// Auto Bagger 
GVL_IO.BG_YFillerTrigger					:= BYTE_TO_BOOL(GVL_IO.OutputsFromHMI[91]);
IF (STATUS.BaggerPrintCmd = 1) THEN 
	MAIN.fbEL6001.M_PrintLabel(isPremium := FALSE);  
    STATUS.BaggerPrintCmd := 0;
    (* We now have a separate button for Clear Out Chute Counts
    Config.PremiumCount1 := 0;
    Config.PremiumCount2 := 0;
	Config.GoodCount1 := 0;
	Config.GoodCount2 := 0;
    *) 
 END_IF // print label trigger from HMI

GVL_IO.BG_YCloseChute1 := BYTE_TO_BOOL(GVL_IO.OutputsFromHMI[92]); 	
GVL_IO.BG_YOpenChute1  := BYTE_TO_BOOL(GVL_IO.OutputsFromHMI[93]);  	
GVL_IO.BG_YCloseChute2 := BYTE_TO_BOOL(GVL_IO.OutputsFromHMI[94]); 	
GVL_IO.BG_YOpenChute2  := BYTE_TO_BOOL(GVL_IO.OutputsFromHMI[95]); 	
GVL_IO.BG_YCloseChute3 := BYTE_TO_BOOL(GVL_IO.OutputsFromHMI[96]); 	
GVL_IO.BG_YOpenChute3  := BYTE_TO_BOOL(GVL_IO.OutputsFromHMI[97]); 	
GVL_IO.BG_YCloseChute4 := BYTE_TO_BOOL(GVL_IO.OutputsFromHMI[98]); 	
GVL_IO.BG_YOpenChute4  := BYTE_TO_BOOL(GVL_IO.OutputsFromHMI[99]); 	






// Reject Unload
GVL_IO.RJ_YRejectPushExtend				:= BYTE_TO_BOOL(GVL_IO.OutputsFromHMI[101]); 	
GVL_IO.RJ_YRejectPushRetract			:= BYTE_TO_BOOL(GVL_IO.OutputsFromHMI[102]); 	
//GVL_IO.RJ_YPalletReleaseExtend			:= BYTE_TO_BOOL(GVL_IO.OutputsFromHMI[103]); 	
//GVL_IO.RJ_YPalletReleaseRetract			:= BYTE_TO_BOOL(GVL_IO.OutputsFromHMI[104]); 	
GVL_IO.RJ_YPalletHoldDownExtend_Home			:= BYTE_TO_BOOL(GVL_IO.OutputsFromHMI[105]); 	
GVL_IO.RJ_YPalletHoldDownRetract_Engage		:= BYTE_TO_BOOL(GVL_IO.OutputsFromHMI[106]); 	
                                                                                        
// Main Control System

GVL_IO.MC_YStackLightYellow				:= BYTE_TO_BOOL(GVL_IO.OutputsFromHMI[111]);
GVL_IO.MC_YStackLightRed				:= BYTE_TO_BOOL(GVL_IO.OutputsFromHMI[112]);
GVL_IO.MC_YStackLightGreen				:= BYTE_TO_BOOL(GVL_IO.OutputsFromHMI[113]);
                                        

// Prime Mover 
GVL_IO.MM_YEnableMagneMotion           := BYTE_TO_BOOL(GVL_IO.OutputsFromHMI[121]);

END_FUNCTION_BLOCK

// ---- POUs/FrameworkPOUs/PrepareInputsDataStructureForHMI.TcPOU
// Fill up the appropriate data structure to send input data to the HMI 
FUNCTION_BLOCK FINAL PrepareInputsDataStructureForHMI
VAR_INPUT
END_VAR
VAR_OUTPUT
END_VAR
VAR
	UL_X: INT;
END_VAR

memset(ADR(GVL_IO.InputsForHMI[1]),0,SIZEOF(GVL_IO.InputsForHMI)); //clear out the input array

// Load Station
GVL_IO.InputsForHMI[1] := 	BOOL_TO_BYTE(GVL_IO.LD_XPalletHoldRetractEngage);
GVL_IO.InputsForHMI[2] := 	BOOL_TO_BYTE(GVL_IO.LD_XPalletHoldDownExtendHome);
GVL_IO.InputsForHMI[3] := 	BOOL_TO_BYTE(GVL_IO.LD_XPalletReleaseHome);
GVL_IO.InputsForHMI[4] := 	BOOL_TO_BYTE(GVL_IO.LD_XPalletReleaseExtended);
GVL_IO.InputsForHMI[15] := 	BOOL_TO_BYTE(GVL_IO.LD_XPalletCloseExtended_1_2);
GVL_IO.InputsForHMI[16] := 	BOOL_TO_BYTE(GVL_IO.LD_XPalletCloseExtended_3_4);
GVL_IO.InputsForHMI[17] := 	BOOL_TO_BYTE(GVL_IO.LD_XPalletCloseRetracted_1_2);
GVL_IO.InputsForHMI[18] := 	BOOL_TO_BYTE(GVL_IO.LD_XPalletCloseRetracted_3_4);

// Yushin Robot 
GVL_IO.InputsForHMI[5] := 	BOOL_TO_BYTE(GVL_IO.YU_XPrepareToLoad);
GVL_IO.InputsForHMI[6] := 	BOOL_TO_BYTE(GVL_IO.YU_XToolUp);           
GVL_IO.InputsForHMI[7] := 	BOOL_TO_BYTE(GVL_IO.YU_XToolDown);
GVL_IO.InputsForHMI[8] := 	BOOL_TO_BYTE(GVL_IO.YU_XLocBit0);
GVL_IO.InputsForHMI[9] := 	BOOL_TO_BYTE(GVL_IO.YU_XLocBit1);

// Burnoff
GVL_IO.InputsForHMI[11] := 	BOOL_TO_BYTE(GVL_IO.BU_XAlarm);

// Ionizer 
GVL_IO.InputsForHMI[12] := 	BOOL_TO_BYTE(GVL_IO.IZ_XIonAlarm);
GVL_IO.InputsForHMI[13] := 	BOOL_TO_BYTE(GVL_IO.IZ_XConditionAlarm);
GVL_IO.InputsForHMI[14] := 	BOOL_TO_BYTE(GVL_IO.IZ_XAlarm);
// borrowing 15,16,17,18 for Load Station Pallet Close inputs
// Vision
GVL_IO.InputsForHMI[21] := 	BOOL_TO_BYTE(GVL_IO.VS_XToolingLocationUpper);
GVL_IO.InputsForHMI[22] := 	BOOL_TO_BYTE(GVL_IO.VS_XRun);
GVL_IO.InputsForHMI[23] := 	BOOL_TO_BYTE(GVL_IO.VS_XReady1);
GVL_IO.InputsForHMI[24] := 	BOOL_TO_BYTE(GVL_IO.VS_XReady2);
GVL_IO.InputsForHMI[25] := 	BOOL_TO_BYTE(GVL_IO.VS_XReady3);
GVL_IO.InputsForHMI[26] := 	BOOL_TO_BYTE(GVL_IO.VS_XReady4);
GVL_IO.InputsForHMI[27] := 	BOOL_TO_BYTE(GVL_IO.VS_XCam1JudgeVal);
GVL_IO.InputsForHMI[28] := 	BOOL_TO_BYTE(GVL_IO.VS_XCam2JudgeVal);
GVL_IO.InputsForHMI[29] := 	BOOL_TO_BYTE(GVL_IO.VS_XCam3JudgeVal);
GVL_IO.InputsForHMI[30] := 	BOOL_TO_BYTE(GVL_IO.VS_XCam4JudgeVal);
GVL_IO.InputsForHMI[92] := 	BOOL_TO_BYTE(GVL_IO.VS_XPartEmpty);
GVL_IO.InputsForHMI[93] :=  BOOL_TO_BYTE(GVL_IO.VS_XToolingLocationLower);
GVL_IO.InputsForHMI[94] :=  BOOL_TO_BYTE(GVL_IO.VS_XPartPresentBeforeVision);

// Piston Insert 
GVL_IO.InputsForHMI[31] := 	BOOL_TO_BYTE(GVL_IO.PI_XPalletHoldDownHome);
GVL_IO.InputsForHMI[32] := 	BOOL_TO_BYTE(GVL_IO.PI_XPalletHoldDownExtended);
GVL_IO.InputsForHMI[33] := 	BOOL_TO_BYTE(GVL_IO.PI_XPistonPresentEscapement);
GVL_IO.InputsForHMI[34] := 	BOOL_TO_BYTE(GVL_IO.PI_XEscapementAtInsertLoc);
GVL_IO.InputsForHMI[35] := 	BOOL_TO_BYTE(GVL_IO.PI_XEscapementAtBowl);
GVL_IO.InputsForHMI[36] := 	BOOL_TO_BYTE(GVL_IO.PI_XToolAt55_10_Barrel);
GVL_IO.InputsForHMI[37] := 	BOOL_TO_BYTE(GVL_IO.PI_XToolAt3_30_Barrel);
GVL_IO.InputsForHMI[38] := 	BOOL_TO_BYTE(GVL_IO.PI_XBarrelHoldDownHome);
GVL_IO.InputsForHMI[39] := 	BOOL_TO_BYTE(GVL_IO.PI_XBarrelHoldDownExtended);

//GVL_IO.InputsForHMI[40] := 1;
GVL_IO.InputsForHMI[40] := BOOL_TO_BYTE(GVL_IO.PI_XMtrOUT0);
GVL_IO.InputsForHMI[41] := BOOL_TO_BYTE(GVL_IO.PI_XMtrOUT1);
GVL_IO.InputsForHMI[42] := BOOL_TO_BYTE(GVL_IO.PI_XMtrBusy);
GVL_IO.InputsForHMI[43] := BOOL_TO_BYTE(GVL_IO.PI_XMtrServoEnabled);
GVL_IO.InputsForHMI[44] := BOOL_TO_BYTE(GVL_IO.PI_XMtrServoHomed);
GVL_IO.InputsForHMI[45] := BOOL_TO_BYTE(GVL_IO.PI_XMtrMoveCompl);
GVL_IO.InputsForHMI[46] := BOOL_TO_BYTE(GVL_IO.PI_XMtrEStopped);
GVL_IO.InputsForHMI[47] := BOOL_TO_BYTE(GVL_IO.PI_XMtrAlarm);


// Cap Insert

GVL_IO.InputsForHMI[56] := 	BOOL_TO_BYTE(GVL_IO.CP_XPalletHoldDownHome);
GVL_IO.InputsForHMI[57] := 	BOOL_TO_BYTE(GVL_IO.CP_XPalletHoldDownExtended);
GVL_IO.InputsForHMI[58] := 	BOOL_TO_BYTE(GVL_IO.CP_XCapSlideRetracted);
GVL_IO.InputsForHMI[59] := 	BOOL_TO_BYTE(GVL_IO.CP_XCapSlideExtended);


// Unload 

GVL_IO.InputsForHMI[77] :=  BOOL_TO_BYTE(GVL_IO.UL_1_XPalletHoldDownRetracted_Engaged);
GVL_IO.InputsForHMI[78] :=  BOOL_TO_BYTE(GVL_IO.UL_1_XPalletHoldDownExtended_Home);
GVL_IO.InputsForHMI[79] := 	BOOL_TO_BYTE(GVL_IO.UL_1_XBarrelPresent);
GVL_IO.InputsForHMI[80] :=  BOOL_TO_BYTE(GVL_IO.UL_2_XPalletHoldDownRetracted_Engaged);
GVL_IO.InputsForHMI[81] :=  BOOL_TO_BYTE(GVL_IO.UL_2_XPalletHoldDownExtended_Home);
GVL_IO.InputsForHMI[82] := 	BOOL_TO_BYTE(GVL_IO.UL_2_XBarrelPresent);
GVL_IO.InputsForHMI[83] :=  BOOL_TO_BYTE(GVL_IO.UL_3_XPalletHoldDownRetracted_Engaged);
GVL_IO.InputsForHMI[84] :=  BOOL_TO_BYTE(GVL_IO.UL_3_XPalletHoldDownExtended_Home);
GVL_IO.InputsForHMI[85] := 	BOOL_TO_BYTE(GVL_IO.UL_3_XBarrelPresent);
GVL_IO.InputsForHMI[86] :=  BOOL_TO_BYTE(GVL_IO.UL_4_XPalletHoldDownRetracted_Engaged);
GVL_IO.InputsForHMI[87] :=  BOOL_TO_BYTE(GVL_IO.UL_4_XPalletHoldDownExtended_Home);
GVL_IO.InputsForHMI[88] := 	BOOL_TO_BYTE(GVL_IO.UL_4_XBarrelPresent);


// bagger
GVL_IO.InputsForHMI[91] := 	BOOL_TO_BYTE(GVL_IO.BG_XBaggerBusy);
//borrowing 92 for vision
// borrowing 93 for vision
// borrow 94 for vision
GVL_IO.InputsForHMI[115] := 	BOOL_TO_BYTE(GVL_IO.BG_XBagsLow);
GVL_IO.InputsForHMI[116] := 	BOOL_TO_BYTE(GVL_IO.BG_XBaggerOKNoFault);
GVL_IO.InputsForHMI[117] := 	BOOL_TO_BYTE(GVL_IO.BG_XBaggerWaitingForLabel);
GVL_IO.InputsForHMI[118] := 	BOOL_TO_BYTE(GVL_IO.BG_XBaggerReadyForFiller);


GVL_IO.InputsForHMI[95] := 	BOOL_TO_BYTE(GVL_IO.BG_XChute1Closed);
GVL_IO.InputsForHMI[96] := 	BOOL_TO_BYTE(GVL_IO.BG_XChute1Open);
GVL_IO.InputsForHMI[97] := 	BOOL_TO_BYTE(GVL_IO.BG_XChute2Closed);
GVL_IO.InputsForHMI[98] := 	BOOL_TO_BYTE(GVL_IO.BG_XChute2Open);
GVL_IO.InputsForHMI[99] := 	BOOL_TO_BYTE(GVL_IO.BG_XChute3Closed);
GVL_IO.InputsForHMI[100] := BOOL_TO_BYTE(GVL_IO.BG_XChute3Open);  
GVL_IO.InputsForHMI[108] := BOOL_TO_BYTE(GVL_IO.BG_XChute4Closed);
GVL_IO.InputsForHMI[109] := BOOL_TO_BYTE(GVL_IO.BG_XChute4Open);  



// Reject Station 
GVL_IO.InputsForHMI[101] := 	BOOL_TO_BYTE(GVL_IO.RJ_XRejectCylinderHome);
GVL_IO.InputsForHMI[102] := 	BOOL_TO_BYTE(GVL_IO.RJ_XRejectCylinderExtended);
//GVL_IO.InputsForHMI[103] := 	BOOL_TO_BYTE(GVL_IO.RJ_XPalletReleaseHome);
//GVL_IO.InputsForHMI[104] := 	BOOL_TO_BYTE(GVL_IO.RJ_XPalletReleaseExtended);
GVL_IO.InputsForHMI[105] := 	BOOL_TO_BYTE(GVL_IO.RJ_XPartPresent);
GVL_IO.InputsForHMI[106] := 	BOOL_TO_BYTE(GVL_IO.RJ_XPalletHoldDownRetracted_Engaged);
GVL_IO.InputsForHMI[107] := 	BOOL_TO_BYTE(GVL_IO.RJ_XPalletHoldDownExtended_Home);
// borrowing 108 and 109 for Autobagger inputs

// Main Control System
GVL_IO.InputsForHMI[111] := 	BOOL_TO_BYTE(GVL_IO.MC_XAirPressureOK);
GVL_IO.InputsForHMI[112] := 	BOOL_TO_BYTE(GVL_IO.MC_XStartPB);
GVL_IO.InputsForHMI[113] := 	BOOL_TO_BYTE(GVL_IO.MC_XStopPB);
GVL_IO.InputsForHMI[114] := 	BOOL_TO_BYTE(GVL_IO.MC_NotEStopped);
// borrowing 115,116,117,118 for bagger inputs

END_FUNCTION_BLOCK

// ---- POUs/FrameworkPOUs/PrepareOutputsDataStructureForHMI.TcPOU
// Fill up the appropriate data structure to send input data to the HMI 
FUNCTION_BLOCK FINAL PrepareOutputsDataStructureForHMI
VAR_INPUT
END_VAR
VAR_OUTPUT
END_VAR
VAR
END_VAR

memset(ADR(GVL_IO.OutputsForHMI[1]),0,SIZEOF(GVL_IO.InputsForHMI)); //clear out the output array

// Load Position Outputs 

GVL_IO.OutputsForHMI[1] 	:= BOOL_TO_BYTE(GVL_IO.LD_YPalletHoldDownRetractEngage);
GVL_IO.OutputsForHMI[2] 	:= BOOL_TO_BYTE(GVL_IO.LD_YPalletHoldDownExtendHome);
GVL_IO.OutputsForHMI[3] 	:= BOOL_TO_BYTE(GVL_IO.LD_YPalletReleaseExtend);
GVL_IO.OutputsForHMI[4] 	:= BOOL_TO_BYTE(GVL_IO.LD_YPalletReleaseRetract);
GVL_IO.OutputsForHMI[8]     := BOOL_TO_BYTE(GVL_IO.LD_YPalletCloseExtend);
GVL_IO.OutputsForHMI[9]     := BOOL_TO_BYTE(GVL_IO.LD_YPalletCloseRetract);

// Yushin Robot Interface Outputs

GVL_IO.OutputsForHMI[5] 	:= BOOL_TO_BYTE(GVL_IO.YU_YOkToLoad);
GVL_IO.OutputsForHMI[6] 	:= BOOL_TO_BYTE(GVL_IO.YU_YAckPartsHeld);
GVL_IO.OutputsForHMI[10]    := BOOL_TO_BYTE(GVL_IO.YU_YIMBADIsOK);

//Ionizer Outputs

GVL_IO.OutputsForHMI[7] 	:= BOOL_TO_BYTE(GVL_IO.IZ_YInterrupt);
//GVL_IO.OutputsForHMI[8]     := BOOL_TO_BYTE(GVL_IO.IZ_YIonizerAirON);
//GVL_IO.OutputsForHMI[9]     := BOOL_TO_BYTE(GVL_IO.IZ_YIonizerAirOFF);
// give 10 to Yushin

// Vision
GVL_IO.OutputsForHMI[21] 	:= BOOL_TO_BYTE(GVL_IO.VS_YBarrelLED);
GVL_IO.OutputsForHMI[22] 	:= BOOL_TO_BYTE(GVL_IO.VS_YCmdRequest);
GVL_IO.OutputsForHMI[23] 	:= BOOL_TO_BYTE(GVL_IO.VS_YResultAck);
GVL_IO.OutputsForHMI[24] 	:= BOOL_TO_BYTE(GVL_IO.VS_YErrorReset);
GVL_IO.OutputsForHMI[25] 	:= BOOL_TO_BYTE(GVL_IO.VS_YTrigger1);
GVL_IO.OutputsForHMI[26] 	:= BOOL_TO_BYTE(GVL_IO.VS_YTrigger2);
GVL_IO.OutputsForHMI[27] 	:= BOOL_TO_BYTE(GVL_IO.VS_YTrigger3);
GVL_IO.OutputsForHMI[28] 	:= BOOL_TO_BYTE(GVL_IO.VS_YTrigger4);


// Piston Insert 
GVL_IO.OutputsForHMI[31] 	:= BOOL_TO_BYTE(GVL_IO.PI_YPalletHoldDownExtend);
GVL_IO.OutputsForHMI[32] 	:= BOOL_TO_BYTE(GVL_IO.PI_YPalletHoldDownRetract);
GVL_IO.OutputsForHMI[33] 	:= BOOL_TO_BYTE(GVL_IO.PI_YEscapementToBowl);
GVL_IO.OutputsForHMI[34] 	:= BOOL_TO_BYTE(GVL_IO.PI_YEscapementToWork);
GVL_IO.OutputsForHMI[35] 	:= BOOL_TO_BYTE(GVL_IO.PI_YBarrelBackupExtend);
GVL_IO.OutputsForHMI[36] 	:= BOOL_TO_BYTE(GVL_IO.PI_YBarrelBackupRetract);
GVL_IO.OutputsForHMI[37] 	:= BOOL_TO_BYTE(GVL_IO.PI_YPistonBowlON);
GVL_IO.OutputsForHMI[38] 	:= BOOL_TO_BYTE(GVL_IO.PI_YPistonBowlOFF);

GVL_IO.OutputsForHMI[40] 	:= BOOL_TO_BYTE(GVL_IO.PI_YMtrStepSelectIN0);
GVL_IO.OutputsForHMI[41] 	:= BOOL_TO_BYTE(GVL_IO.PI_YMtrStepSelectIN1);
GVL_IO.OutputsForHMI[42] 	:= BOOL_TO_BYTE(GVL_IO.PI_YMtrStepSelectIN2);
GVL_IO.OutputsForHMI[43] 	:= BOOL_TO_BYTE(GVL_IO.PI_YMtrHoldMove);
GVL_IO.OutputsForHMI[44] 	:= BOOL_TO_BYTE(GVL_IO.PI_YMtrSetEnable);
GVL_IO.OutputsForHMI[45] 	:= BOOL_TO_BYTE(GVL_IO.PI_YMtrDriveStepTrigger);
GVL_IO.OutputsForHMI[46] 	:= BOOL_TO_BYTE(GVL_IO.PI_YMtrReset);
GVL_IO.OutputsForHMI[47] 	:= BOOL_TO_BYTE(GVL_IO.PI_YMtrGoHome);
GVL_IO.OutputsForHMI[48] 	:= BOOL_TO_BYTE(GVL_IO.PI_YMtrJogNeg);
GVL_IO.OutputsForHMI[49] 	:= BOOL_TO_BYTE(GVL_IO.PI_YMtrJogPos);
GVL_IO.OutputsForHMI[50] 	:= BOOL_TO_BYTE(GVL_IO.PI_YMtrSwitchJogInch);
// Cap Insert 

GVL_IO.OutputsForHMI[57] 	:= BOOL_TO_BYTE(GVL_IO.CP_YCapSlideExtend);
GVL_IO.OutputsForHMI[58] 	:= BOOL_TO_BYTE(GVL_IO.CP_YCapSlideRetract);
GVL_IO.OutputsForHMI[59] 	:= BOOL_TO_BYTE(GVL_IO.CP_YPalletHoldDownExtend);
GVL_IO.OutputsForHMI[60] 	:= BOOL_TO_BYTE(GVL_IO.CP_YPalletHoldDownRetract);


// Good Unload Outputs
 
GVL_IO.OutputsForHMI[71] 	:= BOOL_TO_BYTE(GVL_IO.UL_1_YPalletHoldDownExtend_Home);
GVL_IO.OutputsForHMI[72] 	:= BOOL_TO_BYTE(GVL_IO.UL_1_YPalletHoldDownRetract_Engage);
GVL_IO.OutputsForHMI[73] 	:= BOOL_TO_BYTE(GVL_IO.UL_2_YPalletHoldDownExtend_Home);
GVL_IO.OutputsForHMI[74] 	:= BOOL_TO_BYTE(GVL_IO.UL_2_YPalletHoldDownRetract_Engage);
GVL_IO.OutputsForHMI[75] 	:= BOOL_TO_BYTE(GVL_IO.UL_3_YPalletHoldDownExtend_Home);
GVL_IO.OutputsForHMI[76] 	:= BOOL_TO_BYTE(GVL_IO.UL_3_YPalletHoldDownRetract_Engage);
GVL_IO.OutputsForHMI[77] 	:= BOOL_TO_BYTE(GVL_IO.UL_4_YPalletHoldDownExtend_Home);   
GVL_IO.OutputsForHMI[78] 	:= BOOL_TO_BYTE(GVL_IO.UL_4_YPalletHoldDownRetract_Engage);

GVL_IO.OutputsForHMI[79] 	:= BOOL_TO_BYTE(GVL_IO.UL_1_YRejectPushExtend);
GVL_IO.OutputsForHMI[80] 	:= BOOL_TO_BYTE(GVL_IO.UL_2_YRejectPushExtend);
GVL_IO.OutputsForHMI[81] 	:= BOOL_TO_BYTE(GVL_IO.UL_3_YRejectPushExtend);
GVL_IO.OutputsForHMI[82] 	:= BOOL_TO_BYTE(GVL_IO.UL_4_YRejectPushExtend);

GVL_IO.OutputsForHMI[83] 	:= BOOL_TO_BYTE(GVL_IO.UL_1_YRejectPushRetract);
GVL_IO.OutputsForHMI[84] 	:= BOOL_TO_BYTE(GVL_IO.UL_2_YRejectPushRetract);
GVL_IO.OutputsForHMI[85] 	:= BOOL_TO_BYTE(GVL_IO.UL_3_YRejectPushRetract);
GVL_IO.OutputsForHMI[86] 	:= BOOL_TO_BYTE(GVL_IO.UL_4_YRejectPushRetract);




// Auto Bagger 
GVL_IO.OutputsForHMI[91] 	:= 	BOOL_TO_BYTE(GVL_IO.BG_YFillerTrigger);
GVL_IO.OutputsForHMI[92] 	:= 	BOOL_TO_BYTE(GVL_IO.BG_YCloseChute1);
GVL_IO.OutputsForHMI[93] 	:= 	BOOL_TO_BYTE(GVL_IO.BG_YOpenChute1);
GVL_IO.OutputsForHMI[94] 	:= 	BOOL_TO_BYTE(GVL_IO.BG_YCloseChute2);
GVL_IO.OutputsForHMI[95] 	:= 	BOOL_TO_BYTE(GVL_IO.BG_YOpenChute2);
GVL_IO.OutputsForHMI[96] 	:= 	BOOL_TO_BYTE(GVL_IO.BG_YCloseChute3);
GVL_IO.OutputsForHMI[97] 	:= 	BOOL_TO_BYTE(GVL_IO.BG_YOpenChute3);
GVL_IO.OutputsForHMI[98] 	:= 	BOOL_TO_BYTE(GVL_IO.BG_YCloseChute4);
GVL_IO.OutputsForHMI[99] 	:= 	BOOL_TO_BYTE(GVL_IO.BG_YOpenChute4);



// Reject Unload
GVL_IO.OutputsForHMI[101] 	:= BOOL_TO_BYTE(GVL_IO.RJ_YRejectPushExtend);
GVL_IO.OutputsForHMI[102] 	:= BOOL_TO_BYTE(GVL_IO.RJ_YRejectPushRetract);
//GVL_IO.OutputsForHMI[103] 	:= BOOL_TO_BYTE(GVL_IO.RJ_YPalletReleaseExtend);
//GVL_IO.OutputsForHMI[104] 	:= BOOL_TO_BYTE(GVL_IO.RJ_YPalletReleaseRetract);
GVL_IO.OutputsForHMI[105] 	:= BOOL_TO_BYTE(GVL_IO.RJ_YPalletHoldDownExtend_Home);
GVL_IO.OutputsForHMI[106] 	:= BOOL_TO_BYTE(GVL_IO.RJ_YPalletHoldDownRetract_Engage);

// Main Control System

GVL_IO.OutputsForHMI[111] 	:= BOOL_TO_BYTE(GVL_IO.MC_YStackLightYellow);
GVL_IO.OutputsForHMI[112] 	:= BOOL_TO_BYTE(GVL_IO.MC_YStackLightRed);
GVL_IO.OutputsForHMI[113] 	:= BOOL_TO_BYTE(GVL_IO.MC_YStackLightGreen);



// Prime Mover 
GVL_IO.OutputsForHMI[121] 	:= BOOL_TO_BYTE(GVL_IO.MM_YEnableMagneMotion);

END_FUNCTION_BLOCK

// ---- POUs/FrameworkPOUs/SetOutputsToFieldBus.TcPOU
// Setup the appropriate output from the outputs  coming from the logic (either PLC or HMI) which are not directly addressable in the linking of variables
FUNCTION_BLOCK FINAL SetOutputsToFieldBus
VAR_INPUT
END_VAR
VAR_OUTPUT
END_VAR
VAR
END_VAR

//SMC EX260-SEC Valve Bank 1    
(* Terminal 1*)		GVL_IO.SMCEX260_1_Byte0.0 := GVL_IO.LD_YPalletReleaseExtend;
(* Terminal 2*)		GVL_IO.SMCEX260_1_Byte0.1 := GVL_IO.LD_YPalletReleaseRetract;
(* Terminal 3*)		GVL_IO.SMCEX260_1_Byte0.2 := GVL_IO.LD_YPalletCloseExtend;
(* Terminal 4*)		GVL_IO.SMCEX260_1_Byte0.3 := GVL_IO.LD_YPalletCloseRetract;
(* Terminal 5*)		GVL_IO.SMCEX260_1_Byte0.4 := GVL_IO.LD_YPalletHoldDownExtendHome;
(* Terminal 6*)		GVL_IO.SMCEX260_1_Byte0.5 := GVL_IO.LD_YPalletHoldDownRetractEngage;
(* Terminal 7*)		GVL_IO.SMCEX260_1_Byte0.6 := GVL_IO.PI_YEscapementToBowl;
(* Terminal 8*)		GVL_IO.SMCEX260_1_Byte0.7 := GVL_IO.PI_YEscapementToWork;
					
(* Terminal 9*) 	GVL_IO.SMCEX260_1_Byte1.0 := GVL_IO.PI_YPalletHoldDownExtend; 
(* Terminal 10*)	GVL_IO.SMCEX260_1_Byte1.1 := GVL_IO.PI_YPalletHoldDownRetract;
(* Terminal 11*)	GVL_IO.SMCEX260_1_Byte1.2 := 0;
(* Terminal 12*)	GVL_IO.SMCEX260_1_Byte1.3 := 0;
(* Terminal 13*)	GVL_IO.SMCEX260_1_Byte1.4 := 0;
(* Terminal 14*)	GVL_IO.SMCEX260_1_Byte1.5 := 0;
(* Terminal 15*)	GVL_IO.SMCEX260_1_Byte1.6 := 0;
(* Terminal 16*)	GVL_IO.SMCEX260_1_Byte1.7 := 0;
	
(* Terminal 17*) 	GVL_IO.SMCEX260_1_Byte2.0 :=0;
(* Terminal 18*)	GVL_IO.SMCEX260_1_Byte2.1 :=0;
(* Terminal 19*)	GVL_IO.SMCEX260_1_Byte2.2 :=0;
(* Terminal 20*)	GVL_IO.SMCEX260_1_Byte2.3 :=0;
(* Terminal 21*)	GVL_IO.SMCEX260_1_Byte2.4 :=0;
(* Terminal 22*)	GVL_IO.SMCEX260_1_Byte2.5 :=0;
(* Terminal 23*)	GVL_IO.SMCEX260_1_Byte2.6 :=0;
(* Terminal 24*)	GVL_IO.SMCEX260_1_Byte2.7 :=0;
	
(* Terminal x*) 	GVL_IO.SMCEX260_1_Byte3.0 :=0;
(* Terminal x*)		GVL_IO.SMCEX260_1_Byte3.1 :=0;
(* Terminal x*)		GVL_IO.SMCEX260_1_Byte3.2 :=0;
(* Terminal x*)		GVL_IO.SMCEX260_1_Byte3.3 :=0;
(* Terminal x*)		GVL_IO.SMCEX260_1_Byte3.4 :=0;
(* Terminal x*)		GVL_IO.SMCEX260_1_Byte3.5 :=0;
(* Terminal x*)		GVL_IO.SMCEX260_1_Byte3.6 :=0;
(* Terminal x*)		GVL_IO.SMCEX260_1_Byte3.7 :=0;
						
//SMC EX260-SEC Valve Bank 2
(* Terminal 1*)		GVL_IO.SMCEX260_2_Byte0.0 := GVL_IO.BG_YCloseChute1;
(* Terminal 2*)		GVL_IO.SMCEX260_2_Byte0.1 := GVL_IO.BG_YOpenChute1;
(* Terminal 3*)		GVL_IO.SMCEX260_2_Byte0.2 := GVL_IO.BG_YCloseChute2;
(* Terminal 4*)		GVL_IO.SMCEX260_2_Byte0.3 := GVL_IO.BG_YOpenChute2;
(* Terminal 5*)		GVL_IO.SMCEX260_2_Byte0.4 := GVL_IO.CP_YCapSlideExtend;
(* Terminal 6*)		GVL_IO.SMCEX260_2_Byte0.5 := GVL_IO.CP_YCapSlideRetract;
(* Terminal 7*)		GVL_IO.SMCEX260_2_Byte0.6 := GVL_IO.RJ_YRejectPushRetract;
(* Terminal 8*)		GVL_IO.SMCEX260_2_Byte0.7 := GVL_IO.RJ_YRejectPushExtend;


(* Terminal 9*) 	GVL_IO.SMCEX260_2_Byte1.0 := GVL_IO.RJ_YPalletHoldDownExtend_Home;
(* Terminal 10*)	GVL_IO.SMCEX260_2_Byte1.1 := GVL_IO.RJ_YPalletHoldDownRetract_Engage;
(* Terminal 11*)	GVL_IO.SMCEX260_2_Byte1.2 := GVL_IO.UL_1_YPalletHoldDownExtend_Home;
(* Terminal 12*)	GVL_IO.SMCEX260_2_Byte1.3 := GVL_IO.UL_1_YPalletHoldDownRetract_Engage;
(* Terminal 13*)	GVL_IO.SMCEX260_2_Byte1.4 := GVL_IO.UL_2_YPalletHoldDownExtend_Home;
(* Terminal 14*)	GVL_IO.SMCEX260_2_Byte1.5 := GVL_IO.UL_2_YPalletHoldDownRetract_Engage;
(* Terminal 15*)	GVL_IO.SMCEX260_2_Byte1.6 := GVL_IO.UL_3_YPalletHoldDownExtend_Home;   
(* Terminal 16*)	GVL_IO.SMCEX260_2_Byte1.7 := GVL_IO.UL_3_YPalletHoldDownRetract_Engage;


(* Terminal 17*)	GVL_IO.SMCEX260_2_Byte2.0 := GVL_IO.CP_YPalletHoldDownExtend;
(* Terminal 18*)	GVL_IO.SMCEX260_2_Byte2.1 := GVL_IO.CP_YPalletHoldDownRetract;
(* Terminal 19*)	GVL_IO.SMCEX260_2_Byte2.2 := GVL_IO.UL_4_YPalletHoldDownExtend_Home;   
(* Terminal 20*)	GVL_IO.SMCEX260_2_Byte2.3 := GVL_IO.UL_4_YPalletHoldDownRetract_Engage;
(* Terminal 21*)	GVL_IO.SMCEX260_2_Byte2.4 := GVL_IO.BG_YCloseChute3;
(* Terminal 22*)	GVL_IO.SMCEX260_2_Byte2.5 := GVL_IO.BG_YOpenChute3;
(* Terminal 23*)	GVL_IO.SMCEX260_2_Byte2.6 := GVL_IO.BG_YCloseChute4;
(* Terminal 24*)	GVL_IO.SMCEX260_2_Byte2.7 := GVL_IO.BG_YOpenChute4; 

(* Terminal 25*)	GVL_IO.SMCEX260_2_Byte3.0 := GVL_IO.UL_1_YRejectPushRetract;
(* Terminal 26*)	GVL_IO.SMCEX260_2_Byte3.1 := GVL_IO.UL_1_YRejectPushExtend; 
(* Terminal 27*)	GVL_IO.SMCEX260_2_Byte3.2 := GVL_IO.UL_2_YRejectPushRetract;
(* Terminal 28*)	GVL_IO.SMCEX260_2_Byte3.3 := GVL_IO.UL_2_YRejectPushExtend;
(* Terminal 29*)	GVL_IO.SMCEX260_2_Byte3.4 := GVL_IO.UL_3_YRejectPushRetract;
(* Terminal 30*)	GVL_IO.SMCEX260_2_Byte3.5 := GVL_IO.UL_3_YRejectPushExtend;
(* Terminal 31*)	GVL_IO.SMCEX260_2_Byte3.6 := GVL_IO.UL_4_YRejectPushRetract;
(* Terminal 32*)	GVL_IO.SMCEX260_2_Byte3.7 := GVL_IO.UL_4_YRejectPushExtend;

//(* Terminal 3*)		GVL_IO.SMCEX260_2_Byte0.2 := GVL_IO.CP_YEscapeWallCylinderRetract;
//(* Terminal 4*)		GVL_IO.SMCEX260_2_Byte0.3 := GVL_IO.CP_YEscapeWallCylinderExtend;



//(* Terminal 5*)		GVL_IO.SMCEX260_2_Byte0.4 := GVL_IO.CP_YEscapementToPick;
//(* Terminal 6*)		GVL_IO.SMCEX260_2_Byte0.5 := GVL_IO.CP_YEscapementToBowl;




				            					
//(* Terminal 9*) 	GVL_IO.SMCEX260_2_Byte1.0 := GVL_IO.RJ_YPalletReleaseExtend;
//(* Terminal 10*)	GVL_IO.SMCEX260_2_Byte1.1 := GVL_IO.RJ_YPalletReleaseRetract;
//(* Terminal 12*)	GVL_IO.SMCEX260_2_Byte1.2 := GVL_IO.UL_YPalletReleaseRetract;
//(* Terminal 11*)	GVL_IO.SMCEX260_2_Byte1.3 := GVL_IO.UL_YPalletReleaseExtend;

	               									



//(* Terminal 21*)	GVL_IO.SMCEX260_2_Byte2.4 := GVL_IO.CP_YBarellCenterPinRetract;
//(* Terminal 22*)	GVL_IO.SMCEX260_2_Byte2.5 := GVL_IO.CP_YBarellCenterPinExtend;



	
//////////////////// PISTON INSERT STATION SMC LEY ACTUATOR ETHERNET/IP MAPPING OF DATA 


GVL_IO.SMC_LEY_YUINT0.0 := GVL_IO.PI_YMtrStepSelectIN0;
GVL_IO.SMC_LEY_YUINT0.1 := GVL_IO.PI_YMtrStepSelectIN1;
GVL_IO.SMC_LEY_YUINT0.2 := GVL_IO.PI_YMtrStepSelectIN2;
GVL_IO.SMC_LEY_YUINT0.3 := GVL_IO.PI_YMtrStepSelectIN3;
GVL_IO.SMC_LEY_YUINT0.4 := GVL_IO.PI_YMtrStepSelectIN4;
GVL_IO.SMC_LEY_YUINT0.5 := GVL_IO.PI_YMtrStepSelectIN5;

GVL_IO.SMC_LEY_YUINT0.8  := GVL_IO.PI_YMtrHoldMove;
GVL_IO.SMC_LEY_YUINT0.9  := GVL_IO.PI_YMtrSetEnable;
GVL_IO.SMC_LEY_YUINT0.10 := GVL_IO.PI_YMtrDriveStepTrigger;
GVL_IO.SMC_LEY_YUINT0.11 := GVL_IO.PI_YMtrReset;
GVL_IO.SMC_LEY_YUINT0.12 := GVL_IO.PI_YMtrGoHome;
GVL_IO.SMC_LEY_YUINT0.13 := GVL_IO.PI_YMtrJogNeg;
GVL_IO.SMC_LEY_YUINT0.14 := GVL_IO.PI_YMtrJogPos;
GVL_IO.SMC_LEY_YUINT0.15 := GVL_IO.PI_YMtrSwitchJogInch;
(*
GVL_IO.SMC_LEY_YByte0.0 := GVL_IO.PI_YMtrStepSelectIN0;
GVL_IO.SMC_LEY_YByte0.1 := GVL_IO.PI_YMtrStepSelectIN1;
GVL_IO.SMC_LEY_YByte0.2 := GVL_IO.PI_YMtrStepSelectIN2;
GVL_IO.SMC_LEY_YByte0.3 := GVL_IO.PI_YMtrStepSelectIN3;
GVL_IO.SMC_LEY_YByte0.4 := GVL_IO.PI_YMtrStepSelectIN4;
GVL_IO.SMC_LEY_YByte0.5 := GVL_IO.PI_YMtrStepSelectIN5;

GVL_IO.SMC_LEY_YByte1.0 := GVL_IO.PI_YMtrHoldMove;
GVL_IO.SMC_LEY_YByte1.1 := GVL_IO.PI_YMtrSetEnable;
GVL_IO.SMC_LEY_YByte1.2 := GVL_IO.PI_YMtrDriveStepTrigger;
GVL_IO.SMC_LEY_YByte1.3 := GVL_IO.PI_YMtrReset;
GVL_IO.SMC_LEY_YByte1.4 := GVL_IO.PI_YMtrGoHome;
GVL_IO.SMC_LEY_YByte1.5 := GVL_IO.PI_YMtrJogNeg;
GVL_IO.SMC_LEY_YByte1.6 := GVL_IO.PI_YMtrJogPos;
GVL_IO.SMC_LEY_YByte1.7 := GVL_IO.PI_YMtrSwitchJogInch;
*)

////////////////////// Weiss Pick and Place Mapping EtherCAT ////////////////////////////////////

GVL_IO.UL_YPP_Byte4.0 := GVL_IO.UL_YPP_Enable;
GVL_IO.UL_YPP_Byte4.1 := GVL_IO.UL_YPP_BitA;
GVL_IO.UL_YPP_Byte4.2 := GVL_IO.UL_YPP_BitB;
GVL_IO.UL_YPP_Byte4.3 := GVL_IO.UL_YPP_BitC;
GVL_IO.UL_YPP_Byte4.4 := GVL_IO.UL_YPP_ResetAlarm;
GVL_IO.UL_YPP_Byte4.5 := GVL_IO.UL_YPP_StartHoming;
GVL_IO.UL_YPP_Byte4.6 := GVL_IO.UL_YPP_StartSeq;
GVL_IO.UL_YPP_Byte4.7 := GVL_IO.UL_YPP_Stop;

///////////////////////// Vision Controller ////////////////////////////////////////////////////////

GVL_IO.VS_YByte0.0 := GVL_IO.VS_YCmdRequest;
GVL_IO.VS_YByte0.3 := GVL_IO.VS_YResultAck;
GVL_IO.VS_YByte0.4 := GVL_IO.VS_YErrorReset;

GVL_IO.VS_YByte1.0 := GVL_IO.VS_YTrigger1;
GVL_IO.VS_YByte1.1 := GVL_IO.VS_YTrigger2;
GVL_IO.VS_YByte1.2 := GVL_IO.VS_YTrigger3;
GVL_IO.VS_YByte1.3 := GVL_IO.VS_YTrigger4;
GVL_IO.VS_YByte16 :=  GVL_IO.VS_YCmdNumber;
GVL_IO.VS_YByte20 :=  GVL_IO.VS_YCmdParam1;
GVL_IO.VS_YByte24 :=  GVL_IO.VS_YCmdParam2;

GVL_IO.VS_YBarrelLED_off := NOT GVL_IO.VS_YBarrelLED ;

END_FUNCTION_BLOCK

// ---- POUs/FrameworkPOUs/LotLogging.TcPOU
FUNCTION_BLOCK PUBLIC LotLogging
VAR_INPUT
END_VAR
VAR_OUTPUT
END_VAR
VAR
	PrevLotInProgress : BOOL;
	TimeToLogLot : TON;
END_VAR

IF (NOT LotsData.Lot.LotInProgress) AND PrevLotInProgress THEN
	// create a lot report here and store it
	P_TextModeWriteLot.WriteData := TRUE;	   
END_IF
PrevLotInProgress := LotsData.Lot.LotInProgress;

END_FUNCTION_BLOCK

// ---- POUs/P_TextModeWriteLot.TcPOU
(* Writing of CSV file in text mode. None of the field value is containing any non-printing control characters like line feed, carriage return, quotation marks, semicolon... *)
PROGRAM P_TextModeWriteLot
VAR
	bWrite			: BOOL := FALSE;(* Rising edge starts program execution *)
	sNetId			: T_AmsNetId := '';	(* TwinCAT system network address *)
	sFileName		: T_MaxString := 'C:\LotData.csv';(* CSV destination file path and name *)
	sCSVLine		: T_MaxString := '';(* Single CSV text line (row, record), we are using string as record buffer (your are able to see created fields) *)
	sCSVField		: T_MaxString := '';(* Single CSV field value (column, record field) *)
	bBusy			: BOOL;
	bError			: BOOL;
	nErrId			: UDINT;
	nRow	 		: UDINT 	:= 0;(* Row number (record) *)
	nColumn			: UDINT 	:= 0;(* Column number (record field) *)
	hFile			: UINT		:= 0;(* File handle of the source file *)
	step			: DWORD 	:= 0;
	fbFileOpen		: FB_FileOpen;(* Opens file *)
	fbFileClose		: FB_FileClose;(* Closes file *)
	fbFilePuts		: FB_FilePuts;(* Writes one record (line) *)
	fbWriter		: FB_CSVMemBufferWriter;(* Helper function block used to create CSV data bytes (single record line) *)
	VUT				: BYTE;
	MAX_FIELDS      : BYTE := 15;	

	(*
	
	database		: ARRAY[0..CONFIG.MAX_CSV_ROWS, 0..CONFIG.MAX_CSV_COLUMNS ] OF STRING(CONFIG.MAX_CSV_FIELD_LENGTH) :=[ (* Source PLC database *)
	'0_0', '0_1', '0_2', '0_3', '0_4', '0_5',
	'1_0', '1_1', '1_2', '1_3', '1_4', '1_5',
	'2_0', '2_1', '2_2', '2_3', '2_4', '2_5',
	'3_0', '3_1', '3_2', '3_3', '3_4', '3_5',
	'4_0', '4_1', '4_2', '4_3', '4_4', '4_5',
	'5_0', '5_1', '5_2', '5_3', '5_4', '5_5'];
   *)
	TotalStainArea: REAL := 0;
	TotalStainCount: REAL := 0;
	byCounter : BYTE := 0;
	TotalGood : DINT :=0;
	TotalBad : DINT := 0;
	TotalPremium : DINT :=0;
	cavitycounter: BYTE;
END_VAR

DEFAULT_CSV_FIELD_SEP := 16#2C;(* Comma ASCII code *)
CASE step OF
	0:	(* Wait for rising edge at bWrite variable *)
		IF bWrite THEN
			bWrite 	:= FALSE;
			bBusy 	:= TRUE;
			bError	:= FALSE;
			nErrId	:= 0;
			hFile	:= 0;
			nRow	:= 0;
			nColumn	:= 0;
			step 	:= 1;
		END_IF

	1:	(* Open source file *)
		fbFileOpen(  bExecute := FALSE  );
		fbFileOpen( sNetId := sNetId, sPathName := sFileName, nMode := FOPEN_MODEAPPEND OR FOPEN_MODETEXT,(* Open file in TEXT mode! *)
					ePath := PATH_GENERIC, bExecute := TRUE );
		step := 2;

	2:(* Wait until open not busy *)
		fbFileOpen( bExecute := FALSE, bError => bError, nErrID => nErrID, hFile => hFile );
		IF NOT fbFileOpen.bBusy THEN
			IF NOT fbFileOpen.bError THEN
				step := 3;
			ELSE(* Error: file not found? *)
				step := 100;
			END_IF
		END_IF

	3:(* Convert one PLC record to CSV format *)
	    TotalGood := 0;
		TotalBad := 0;
		TotalPremium := 0;
		FOR byCounter := 1 TO CONFIG.MAX_CAVITY BY 1 DO
			TotalGood := TotalGood + LotsData.Lot.CavityCounts[byCounter].GoodCount;
			TotalBad := TotalBad + LotsData.Lot.CavityCounts[byCounter].BadCount;
			TotalPremium := TotalPremium + LotsData.Lot.CavityCounts[byCounter].GoodCount;
	    END_FOR	
        sCSVLine := '';
		fbWriter.eCmd := eEnumCmd_First;(* Write first field value *)
		IF nRow <= CONFIG.MAX_CSV_ROWS THEN
			FOR nColumn:= 1 TO MAX_FIELDS BY 1 DO
				CASE nColumn OF 
					1: sCSVField := CONCAT( LotsData.Lot.PartNumber,',');  // Part Number
					2: sCSVField := CONCAT( LotsData.Lot.LotNumber,',');  //  Lot Number
					3: sCSVField := CONCAT( LotsData.Lot.JobNumber,','); 
					4: sCSVField := CONCAT( LotsData.Lot.LotDate,',');
					5: sCSVField := CONCAT( LotsData.Lot.PistonLotNumber,','); 
					6: sCSVField := CONCAT( LotsData.Lot.PistonPartNumber,','); 
					7: sCSVField := CONCAT( LotsData.Lot.CapLotNumber,','); 
					8: sCSVField := CONCAT( LotsData.Lot.CapPartNumber,','); 
					9: sCSVField := CONCAT( LotsData.Lot.RawMaterialLotNumber,','); 
					10: sCSVField := CONCAT( LotsData.Lot.BlackConPartNumber,','); 
					11: sCSVField := CONCAT( LotsData.Lot.Comment,','); 					
					12: CASE  LotsData.Lot.BarrelSize OF                                     // Barrel Type
						   	eBarrelType.Size55cc: sCSVField := CONCAT('55cc',',');
						   	eBarrelType.Size30cc: sCSVField := CONCAT('30cc',',');
	 						eBarrelType.Size10cc: sCSVField := CONCAT('10cc',',');
	 						eBarrelType.Size5cc:  sCSVField := CONCAT('5cc',',');
	 						eBarrelType.Size3cc:  sCSVField := CONCAT('3cc',',');
					   END_CASE
					13: sCSVField := CONCAT( DINT_TO_STRING(TotalPremium),','); 
					14: sCSVField := CONCAT( DINT_TO_STRING(TotalGood),','); 
					15: sCSVField := CONCAT( DINT_TO_STRING(TotalBad),','); 
							
					ELSE;
				END_CASE			
			    (* Add new field to the record buffer *)
				fbWriter( 	pBuffer := ADR( sCSVLine ), cbBuffer := SIZEOF( sCSVLine ) - 1, putValue := sCSVField, pValue := 0, cbValue := 0,
							bCRLF := ( nColumn = MAX_FIELDS ) );(* bCRLF == TRUE => Write CRLF after the last field value *)
				IF fbWriter.bOk THEN
					fbWriter.eCmd := eEnumCmd_Next;(* Write next field value *)
				ELSE(* Error *)
					step := 100;
					RETURN;
				END_IF		
			END_FOR
					
			(* FB_FilePuts adds allready CR (carriage return) to the written line.
			We have to replace the $R$L characters with $L character to avoid double CR. *)
			IF RIGHT( sCSVLine, 2 ) = '$R$L' THEN
				sCSVLine := REPLACE( sCSVLine, '$L', 2, LEN( sCSVLine ) - 1 );
			END_IF

			nRow := nRow + 1;(* Increment number of created records (rows) *)
			step := 4;(* Write record to the file *)

		ELSE(* All rows written => Close file *)
			step := 10;
		END_IF

	4:	(* Write single text line *)
		fbFilePuts( bExecute := FALSE );
		fbFilePuts( sNetId := sNetId, hFile := hFile, sLine := sCSVLine, bExecute := TRUE );
		step := 5;

	5:(* Wait until write not busy *)
		fbFilePuts( bExecute := FALSE, bError => bError, nErrID => nErrID );
		IF NOT fbFilePuts.bBusy THEN
			IF NOT fbFilePuts.bError THEN
				step := 10;(* We don't have a next record *)
			ELSE(* Error *)
				step := 100;
			END_IF
		END_IF

	10:	(* Close source file *)
		fbFileClose( bExecute := FALSE );
		fbFileClose( sNetId := sNetId, hFile := hFile, bExecute := TRUE );
		sCSVLine := '';
		step := 11;

	11:(* Wait until close not busy *)
		fbFileClose( bExecute := FALSE, bError => bError, nErrID => nErrID );
		IF ( NOT fbFileClose.bBusy ) THEN
			hFile := 0;
			step := 100;
		END_IF

	100: (* Error or ready step => cleanup *)
		IF ( hFile <> 0 ) THEN
			step := 10; (* Close the source file *)
		ELSE
			bBusy := FALSE;
			step := 0;	(* Ready *)
			// reset all the Lot related information
			FOR cavitycounter:=1 TO CONFIG.MAX_CAVITY BY 1 DO
				LotsData.Lot.CavityCounts[cavitycounter].BadCount :=0;	
				LotsData.Lot.CavityCounts[cavitycounter].GoodCount :=0;	
				LotsData.Lot.CavityCounts[cavitycounter].PremiumCount :=0;	
				LotsData.Lot.CavityCounts[cavitycounter].TotalCount :=0;	
			END_FOR
			LotsData.Lot.LotNumber := 'START NEW LOT';
			LotsData.Lot.JobNumber := '';
			LotsData.Lot.PartNumber := '';				
		END_IF

END_CASE

PROPERTY PUBLIC VehicleID : BYTE
SET
VUT := VehicleID;
END_SET
END_PROPERTY

PROPERTY PUBLIC WriteData : BOOL
SET
bWrite := WriteData;
END_SET
END_PROPERTY

END_PROGRAM

// ---- POUs/FrameworkPOUs/FB_SerialCom.TcPOU
FUNCTION_BLOCK FB_SerialCom
VAR_IN_OUT
	TxBuffer	: ComBuffer;
	RxBuffer	: ComBuffer;
END_VAR
VAR
	Timer		: TON := (PT:=T#1S);
	fbSend		: SendString255;
	bSendBusy	: BOOL;
	eSendErrorID: ComError_t;
    wYear : WORD;
	sYear : STRING;
	wMonth : WORD;
	wDay : WORD;
	wDOY : WORD;
	fbReceive		: ReceiveString;
	sReceivedString	: STRING;
	sLastReceivedString: STRING;
	bStringReceived	: BOOL;
	bReceiveBusy	: BOOL;
	bReceiveError	: BOOL;
	eReceiveErrorID	: ComError_t;
	bReceiveTimeout	: BOOL;
	nReceiveCounter	: UDINT;
	step			: DWORD 	:= 0;
	bPrint			: BOOL := FALSE;(* Rising edge starts program execution *)
	sCSVField		: T_MaxString := '';
	bPremium        : BOOL := FALSE;
END_VAR

// Call the send block every second to repeat the transmission.
// Also call the block as long as it is busy to finish a transmission.
CASE step OF
	0:
		IF bPrint THEN 
			step := 1;
			sCSVField :='';
		END_IF	
	
   
		
	1:  
	    sCSVField := CONCAT('A2>',LotsData.Lot.PartNumber);		
		sCSVField := CONCAT(sCSVField,'$R$L');  // Part Number
		step := 2;		
		bPrint := TRUE;
		//sCSVField := '$01$2A';
	
	2:	
		IF bPrint OR fbSend.Busy THEN
			fbSend(	SendString:= sCSVField,
					TXbuffer:= TxBuffer,
					Busy=> bSendBusy,
					Error=> );			
            bPrint := FALSE;			
			IF fbSend.Error <> COMERROR_NOERROR THEN
				eSendErrorID := fbSend.Error;
			END_IF
		ELSE 
            step := 3;	// done printing // skipping 3 AND 4 here 
			sCSVField :='';
			bPrint := TRUE;
		END_IF
		
	  3: 
        sCSVField := CONCAT('A2>',LotsData.Lot.PartDescription); // Description
		IF (bPremium) THEN
			sCSVField := CONCAT(sCSVField, '-P'); 
		ELSE
			sCSVField := CONCAT(sCSVField, '-G'); 	
		END_IF
		sCSVField := CONCAT(sCSVField, '$R$L'); 
        step := 4;	
		
	4: 
	    IF bPrint OR fbSend.Busy THEN
			fbSend(	SendString:= sCSVField,
					TXbuffer:= TxBuffer,
					Busy=> bSendBusy,
					Error=> );			
            bPrint := FALSE;			
			IF fbSend.Error <> COMERROR_NOERROR THEN
				eSendErrorID := fbSend.Error;
			END_IF
		ELSE 
            step := 5;	// done printing
			sCSVField :='';
			bPrint := TRUE;
		END_IF	
	
    5: 
	   sCSVField := CONCAT('A2>',LotsData.Lot.PistonLotNumber); // Piston Lot Number
	//   sCSVField := CONCAT(sCSVField,' , C Lot #: '); // Piston Lot Number
	 //  sCSVField := CONCAT(sCSVField,LotsData.Lot.CapLotNumber); // Cap Lot Number
       sCSVField := CONCAT(sCSVField, '$R$L'); 	    
	   step := 6;
	 
	 6: 
	    IF bPrint OR fbSend.Busy THEN
			fbSend(	SendString:= sCSVField,
					TXbuffer:= TxBuffer,
					Busy=> bSendBusy,
					Error=> );			
            bPrint := FALSE;			
			IF fbSend.Error <> COMERROR_NOERROR THEN
				eSendErrorID := fbSend.Error;
			END_IF
		ELSE 
            step := 7;	// done printing
			sCSVField :='';
			bPrint := TRUE;
		END_IF	
		
	7:
		sCSVField := CONCAT('A2>',LotsData.Lot.LotNumber ); // Lot Number
        sCSVField := CONCAT(sCSVField,'$R$L');  		 
		step := 8;     
		
	8: 
	    IF bPrint OR fbSend.Busy THEN
			fbSend(	SendString:= sCSVField,
					TXbuffer:= TxBuffer,
					Busy=> bSendBusy,
					Error=> );			
            bPrint := FALSE;			
			IF fbSend.Error <> COMERROR_NOERROR THEN
				eSendErrorID := fbSend.Error;
			END_IF
		ELSE 
            step := 9;	// done printing
			sCSVField :='';
			bPrint := TRUE;
		END_IF
	
	9:
	    wMonth := Logging.fbCurrTime.systemTime.wMonth;
		wYear := Logging.fbCurrTime.systemTime.wYear;
		sYear := WORD_TO_STRING(wYear);
		wDay := Logging.fbCurrTime.systemTime.wDay;
		wDOY := F_GetDOYofYearMonthDay(wYear, wMonth, wDay);
		sCSVField := WORD_TO_STRING(wDOY);
		sCSVField := CONCAT(RIGHT(sYear,1),sCSVField);
		sCSVField := CONCAT('A2>',sCSVField);
       	//sCSVField := CONCAT('A1>','7200'); // replace this with Julian code programmatically	
        sCSVField := CONCAT(sCSVField, '$R$L'); 		 
	    step := 10;
	
    10: 
	    IF bPrint OR fbSend.Busy THEN
			fbSend(	SendString:= sCSVField,
					TXbuffer:= TxBuffer,
					Busy=> bSendBusy,
					Error=> );			
            bPrint := FALSE;			
			IF fbSend.Error <> COMERROR_NOERROR THEN
				eSendErrorID := fbSend.Error;
			END_IF
		ELSE 
            step := 0; //13;	// done printing
			sCSVField :='';			
			bPrint := FALSE;
		END_IF
     
	  
      11: 
	    sCSVField := CONCAT('A1>',LotsData.Lot.CapLotNumber); // Cap Lot Number
		sCSVField := CONCAT(sCSVField, '$R$L'); 	    
		
        step := 10;
       
	 12: 
	    IF bPrint OR fbSend.Busy THEN
			fbSend(	SendString:= sCSVField,
					TXbuffer:= TxBuffer,
					Busy=> bSendBusy,
					Error=> );			
            bPrint := FALSE;			
			IF fbSend.Error <> COMERROR_NOERROR THEN
				eSendErrorID := fbSend.Error;
			END_IF
		ELSE 
            step := 11;	// done printing
			sCSVField :='';
			bPrint := TRUE;
		END_IF
       
	
	
	13:
		sCSVField := CONCAT('rDMXFRM','$R$L'); 		
		step := 14;	
	14:
	 	IF bPrint OR fbSend.Busy THEN
			fbSend(	SendString:= sCSVField,
					TXbuffer:= TxBuffer,
					Busy=> bSendBusy,
					Error=> );			
            bPrint := FALSE;			
			IF fbSend.Error <> COMERROR_NOERROR THEN
				eSendErrorID := fbSend.Error;
			END_IF
		ELSE 
            step := 21;	// done printing finally			
		END_IF
	
	21:
	 	//sCSVField := ('$02L$R$L'); // <STX>L 		
		//sCSVField := CONCAT(sCSVField,'rDMXFRMA1$R$L');  // Recall Label
		sCSVField := 'rDMXFRMA1$R$L';  // Recall Label
		//sCSVField := CONCAT(sCSVField,'E$R$L');  // Terminate label format		
        step := 22;
        bPrint := TRUE;		
    22:
	    IF bPrint OR fbSend.Busy THEN
			fbSend(	SendString:= sCSVField,
					TXbuffer:= TxBuffer,
					Busy=> bSendBusy,
					Error=> );			
            bPrint := FALSE;			
			IF fbSend.Error <> COMERROR_NOERROR THEN
				eSendErrorID := fbSend.Error;
			END_IF
		ELSE 
            step := 0;	// done printing
			sCSVField :='';
			bPrint := TRUE;
		END_IF	
		
	
END_CASE

fbReceive(
	Timeout:= T#1S,
	ReceivedString:= sReceivedString,
	RXbuffer:= RxBuffer,
	StringReceived=> bStringReceived,
	Busy=> bReceiveBusy,
	Error=> ,
	RxTimeout=> bReceiveTimeout );
IF fbReceive.Error <> COMERROR_NOERROR THEN
	eReceiveErrorID := fbReceive.Error;
END_IF
IF bStringReceived THEN
	nReceiveCounter := nReceiveCounter + 1;
	sLastReceivedString := sReceivedString;
END_IF

METHOD PUBLIC M_PrintLabel : BOOL
VAR_INPUT
	isPremium : BOOL;
END_VAR
IF (step =0) THEN
	bPremium := isPremium;
	bPrint := TRUE;
END_IF
END_METHOD

END_FUNCTION_BLOCK

// ---- POUs/P_TextModeWrite.TcPOU
(* Writing of CSV file in text mode. None of the field value is containing any non-printing control characters like line feed, carriage return, quotation marks, semicolon... *)
PROGRAM P_TextModeWrite
VAR
	bWrite			: BOOL := FALSE;(* Rising edge starts program execution *)
	sNetId			: T_AmsNetId := '';	(* TwinCAT system network address *)
	sFileName		: T_MaxString := 'C:\PartsData3.csv';(* CSV destination file path and name *)
	sCSVLine		: T_MaxString := '';(* Single CSV text line (row, record), we are using string as record buffer (your are able to see created fields) *)
	sCSVField		: T_MaxString := '';(* Single CSV field value (column, record field) *)
	bBusy			: BOOL;
	bError			: BOOL;
	nErrId			: UDINT;
	nRow	 		: UDINT 	:= 0;(* Row number (record) *)
	nColumn			: UDINT 	:= 0;(* Column number (record field) *)
	hFile			: UINT		:= 0;(* File handle of the source file *)
	step			: DWORD 	:= 0;
	fbFileOpen		: FB_FileOpen;(* Opens file *)
	fbFileClose		: FB_FileClose;(* Closes file *)
	fbFilePuts		: FB_FilePuts;(* Writes one record (line) *)
	fbWriter		: FB_CSVMemBufferWriter;(* Helper function block used to create CSV data bytes (single record line) *)
	VUT				: BYTE;
	MAX_FIELDS      : BYTE := 22;	

	(*
	
	database		: ARRAY[0..CONFIG.MAX_CSV_ROWS, 0..CONFIG.MAX_CSV_COLUMNS ] OF STRING(CONFIG.MAX_CSV_FIELD_LENGTH) :=[ (* Source PLC database *)
	'0_0', '0_1', '0_2', '0_3', '0_4', '0_5',
	'1_0', '1_1', '1_2', '1_3', '1_4', '1_5',
	'2_0', '2_1', '2_2', '2_3', '2_4', '2_5',
	'3_0', '3_1', '3_2', '3_3', '3_4', '3_5',
	'4_0', '4_1', '4_2', '4_3', '4_4', '4_5',
	'5_0', '5_1', '5_2', '5_3', '5_4', '5_5'];
	
   *)
	//TotalStainArea: REAL := 0;
	TotalStainCount: REAL := 0;
END_VAR

DEFAULT_CSV_FIELD_SEP := 16#2C;(* Comma ASCII code *)
CASE step OF
	0:	(* Wait for rising edge at bWrite variable *)
		IF bWrite THEN
			bWrite 	:= FALSE;
			bBusy 	:= TRUE;
			bError	:= FALSE;
			nErrId	:= 0;
			hFile	:= 0;
			nRow	:= 0;
			nColumn	:= 0;
			step 	:= 1;
		END_IF

	1:	(* Open source file *)
		fbFileOpen(  bExecute := FALSE  );
		fbFileOpen( sNetId := sNetId, sPathName := sFileName, nMode := FOPEN_MODEAPPEND OR FOPEN_MODETEXT,(* Open file in TEXT mode! *)
					ePath := PATH_GENERIC, bExecute := TRUE );
		step := 2;

	2:(* Wait until open not busy *)
		fbFileOpen( bExecute := FALSE, bError => bError, nErrID => nErrID, hFile => hFile );
		IF NOT fbFileOpen.bBusy THEN
			IF NOT fbFileOpen.bError THEN
				step := 3;
			ELSE(* Error: file not found? *)
				step := 100;
			END_IF
		END_IF

	3:(* Convert one PLC record to CSV format *)
		sCSVLine := '';
		fbWriter.eCmd := eEnumCmd_First;(* Write first field value *)
		IF nRow <= CONFIG.MAX_CSV_ROWS THEN
			FOR nColumn:= 1 TO MAX_FIELDS BY 1 DO
				CASE nColumn OF 
					1: sCSVField := CONCAT( PartsData.Status[VUT].PartNumber,',');  // Part Number
					2: sCSVField := CONCAT( PartsData.Status[VUT].LotNumber,',');  //  Lot Number
					3: sCSVField := CONCAT( LotsData.Lot.JobNumber,','); 
					4: sCSVField := CONCAT( LotsData.Lot.LotDate,',');
				//	5: sCSVField := CONCAT( LotsData.Lot.PistonLotNumber,','); 
				//	6: sCSVField := CONCAT( LotsData.Lot.PistonPartNumber,','); 
				//	7: sCSVField := CONCAT( LotsData.Lot.CapLotNumber,','); 
				//	8: sCSVField := CONCAT( LotsData.Lot.CapPartNumber,','); 
				//	9: sCSVField := CONCAT( LotsData.Lot.RawMaterialLotNumber,','); 
				//	10: sCSVField := CONCAT( LotsData.Lot.BlackConPartNumber,','); 
				//	11: sCSVField := CONCAT( LotsData.Lot.Comment,','); 					
					//5: sCSVField := CONCAT( PartsData.Status[VUT].LoadTime,',');  // Load Time  
				    5: sCSVField := CONCAT (PartsData.Status[VUT].VisionInspectTime, ','); //Vision Inspect Time
			//		5: sCSVField := CONCAT (PartsData.Status[VUT].PistonInsertTime, ','); //Piston Insert Time
			//		6: sCSVField := CONCAT (PartsData.Status[VUT].CapInsertTime, ','); //Cap Insert Time
			//		7: sCSVField := CONCAT (PartsData.Status[VUT].UnloadTime, ','); //Good Unload  Time
			//		8: sCSVField := CONCAT (PartsData.Status[VUT].RejectUnloadTime, ','); //Reject Unload Time
					6: sCSVField := CONCAT( INT_TO_STRING(PartsData.Status[VUT].CavityNumber),',');  // Cavity Number
					7: CASE  PartsData.Status[VUT].BarrelSize OF                                     // Barrel Type
						   	eBarrelType.Size55cc: sCSVField := CONCAT('55cc',',');
						   	eBarrelType.Size30cc: sCSVField := CONCAT('30cc',',');
	 						eBarrelType.Size10cc: sCSVField := CONCAT('10cc',',');
	 						eBarrelType.Size5cc:  sCSVField := CONCAT('5cc',',');
	 						eBarrelType.Size3cc:  sCSVField := CONCAT('3cc',',');
					   END_CASE
					8: IF (PartsData.Status[VUT].VisionPass) THEN sCSVField := CONCAT('OK',','); ELSE sCSVField := CONCAT('NG',','); END_IF  // Vision Pass or Fail/Disabled
					9: IF (PartsData.Status[VUT].PistonPass) THEN sCSVField := CONCAT('OK',','); ELSE sCSVField := CONCAT('NG',','); END_IF  // Piston Pass or Fail/Disabled
					10: IF (PartsData.Status[VUT].CapPass) THEN sCSVField := CONCAT('OK',','); ELSE sCSVField := CONCAT('NG',','); END_IF  // Piston Pass or Fail/Disabled
					11: IF (PartsData.Status[VUT].GoodUnload) THEN sCSVField := CONCAT('OK',','); ELSE sCSVField := CONCAT('NG',','); END_IF  // Piston Pass or Fail/Disabled
					12: sCSVField := CONCAT( REAL_TO_STRING(PartsData.Status[VUT].BurnOffTemp),',');  // Burn Off Temperature
					13: sCSVField := CONCAT( REAL_TO_STRING(PartsData.Status[VUT].VisionData.MaxIndividualStainArea),',');  // Piston Stroke
					//13: sCSVField := CONCAT( REAL_TO_STRING(PartsData.Status[VUT].PistonStroke),',');  // Piston Stroke
					//12: ;//sCSVField := CONCAT( REAL_TO_STRING(PartsData.Status[VUT].CapTorque),',');  // Cap Torque
					14: IF (PartsData.Status[VUT].Premium) THEN sCSVField := CONCAT('PREM',','); 
                        ELSIF (PartsData.Status[VUT].Good) THEN sCSVField := CONCAT('GOOD',',');
                        ELSE sCSVField := CONCAT('NG',','); END_IF  // Premium 
					15: IF (NOT PartsData.Status[VUT].VisionData.Cam1Judgement) THEN sCSVField := CONCAT('SSOK',','); ELSE sCSVField := CONCAT('SSNG',','); END_IF  // Short Shot
					16: IF (NOT PartsData.Status[VUT].VisionData.Cam2Judgement) THEN sCSVField := CONCAT('ST2OK ',','); ELSE sCSVField := CONCAT('ST2NG',','); END_IF  // Cam 2 
					17: IF (NOT PartsData.Status[VUT].VisionData.Cam3Judgement) THEN sCSVField := CONCAT('ST3Ok ',','); ELSE sCSVField := CONCAT('ST3NG',','); END_IF  // Cam 3
					18: IF (NOT PartsData.Status[VUT].VisionData.Cam4Judgement) THEN sCSVField := CONCAT('ST4OK',','); ELSE sCSVField := CONCAT('ST4NG',','); END_IF  // Cam 4					
					19:	TotalStainCount  := PartsData.Status[VUT].VisionData.UpperFlawCountCam2 + PartsData.Status[VUT].VisionData.LowerFlawCountCam2 +  					   
						PartsData.Status[VUT].VisionData.UpperFlawCountCam3 + PartsData.Status[VUT].VisionData.LowerFlawCountCam3 +    
						PartsData.Status[VUT].VisionData.UpperFlawCountCam4 + PartsData.Status[VUT].VisionData.LowerFlawCountCam4 ;
						IF (TotalStainCount = 1) THEN
							PartsData.Status[VUT].VisionData.MinIndividualStainArea := PartsData.Status[VUT].VisionData.ModifiedMaxStain;
						END_IF
						sCSVField := CONCAT( REAL_TO_STRING(PartsData.Status[VUT].VisionData.MinIndividualStainArea),',');  
					//Curvature correction math gets applied to Max individual stain but not Min individual stain.  If there is only 1 stain, 
					//Nordson would be confused because Min and Max would not match even though they are the same stain.  To avoid this, if
					//there is only 1 stain I copy the value of the Max stain into the Min stain field.  
						
					20: sCSVField := CONCAT( REAL_TO_STRING(PartsData.Status[VUT].VisionData.ModifiedMaxStain),',');  
					21: sCSVField := CONCAT( REAL_TO_STRING(PartsData.Status[VUT].VisionData.ModifiedStainArea),',');
					//21:
					//	TotalStainArea   := (PartsData.Status[VUT].VisionData.UpperFlawAreaCam2 + PartsData.Status[VUT].VisionData.LowerFlawAreaCam2 + 
					//	PartsData.Status[VUT].VisionData.UpperFlawAreaCam3 + PartsData.Status[VUT].VisionData.LowerFlawAreaCam3 + 
					//	PartsData.Status[VUT].VisionData.UpperFlawAreaCam4 + PartsData.Status[VUT].VisionData.LowerFlawAreaCam4)/1000 ;  
					//    sCSVField := CONCAT( REAL_TO_STRING(TotalStainArea),',');  // Total Stain Area
					22:
                        sCSVField := CONCAT( REAL_TO_STRING(TotalStainCount),',');  // Total Stain Count			
					ELSE;
				END_CASE			
			    (* Add new field to the record buffer *)
				fbWriter( 	pBuffer := ADR( sCSVLine ), cbBuffer := SIZEOF( sCSVLine ) - 1, putValue := sCSVField, pValue := 0, cbValue := 0,
							bCRLF := ( nColumn = MAX_FIELDS ) );(* bCRLF == TRUE => Write CRLF after the last field value *)
				IF fbWriter.bOk THEN
					fbWriter.eCmd := eEnumCmd_Next;(* Write next field value *)
				ELSE(* Error *)
					step := 100;
					RETURN;
				END_IF		
			END_FOR
					
			(* FB_FilePuts adds allready CR (carriage return) to the written line.
			We have to replace the $R$L characters with $L character to avoid double CR. *)
			IF RIGHT( sCSVLine, 2 ) = '$R$L' THEN
				sCSVLine := REPLACE( sCSVLine, '$L', 2, LEN( sCSVLine ) - 1 );
			END_IF

			nRow := nRow + 1;(* Increment number of created records (rows) *)
			step := 4;(* Write record to the file *)
			fbFilePuts( bExecute := FALSE );

		ELSE(* All rows written => Close file *)
			step := 10;
		END_IF

	4:	(* Write single text line *)
		fbFilePuts( bExecute := FALSE );
		fbFilePuts( sNetId := sNetId, hFile := hFile, sLine := sCSVLine, bExecute := TRUE );
		step := 5;

	5:(* Wait until write not busy *)
		fbFilePuts( bExecute := FALSE, bError => bError, nErrID => nErrID );
		IF NOT fbFilePuts.bBusy THEN
			IF NOT fbFilePuts.bError THEN
				step := 10;(* We don't have a next record *)
			ELSE(* Error *)
				step := 100;
			END_IF
		END_IF

	10:	(* Close source file *)
		fbFileClose( bExecute := FALSE );
		fbFileClose( sNetId := sNetId, hFile := hFile, bExecute := TRUE );
		step := 11;

	11:(* Wait until close not busy *)
		fbFileClose( bExecute := FALSE, bError => bError, nErrID => nErrID );
		IF ( NOT fbFileClose.bBusy ) THEN
			hFile := 0;
			step := 100;
		END_IF

	100: (* Error or ready step => cleanup *)
		IF ( hFile <> 0 ) THEN
			step := 10; (* Close the source file *)
		ELSE
			bBusy := FALSE;
			step := 0;	(* Ready *)
		END_IF

END_CASE

PROPERTY PUBLIC CurrWriteStep : DWORD
GET
CurrWriteStep := step;
END_GET
END_PROPERTY

PROPERTY PUBLIC VehicleID : BYTE
SET
VUT := VehicleID;
END_SET
END_PROPERTY

PROPERTY PUBLIC WriteData : BOOL
SET
bWrite := WriteData;
END_SET
END_PROPERTY

END_PROGRAM

// ---- POUs/FrameworkPOUs/BackgroundEL.TcPOU
PROGRAM BackgroundEL
VAR
	(* background communication with the EL6001 terminal *)
	fbEL6001Ctrl		: SerialLineControl;
	bEL6001CtrlError	: BOOL;
	eEL6001CtrlErrorID	: ComError_t;
	(* 	I/O variables for a EL6001 terminal*)
	stIn_EL6001 AT %I*	: EL6inData22B;	(* linked to the EL6001 in the TwinCAT System Manager *)
	stOut_EL6001 AT %Q*	: EL6outData22B;(* linked to the EL6001 in the TwinCAT System Manager *)
END_VAR

(*
The SerialLineControl function block is supposed to be called in every PLC cycle.
It communicates with the serial line hardware device and transmits or receives data.
The SerialLineControl can be called in the standard task (e.g.for PcCOM port usage) 
or in a separate fast task (e.g.for terminal usage) as well.
A fast separate task will be necessary at high baud rates or with KL6001 terminals 
which have a small process image (3 or 5 data bytes only)
*)

(* background communication with the EL6001 terminal *)
fbEL6001Ctrl(
	Mode:= SERIALLINEMODE_EL6_22B, 
	pComIn:= ADR(stIn_EL6001), 
	pComOut:= ADR(stOut_EL6001), 
	SizeComIn:= SIZEOF(stIn_EL6001), 
	Error=> , 
	ErrorID=> , 
	TxBuffer:= GVL_IO.TxBufferEL, 
	RxBuffer:= GVL_IO.RxBufferEL );
IF fbEL6001Ctrl.Error THEN
	bEL6001CtrlError := TRUE;
	eEL6001CtrlErrorID := fbEL6001Ctrl.ErrorID;
END_IF

END_PROGRAM

// ---- POUs/FrameworkPOUs/EventMsg.TcPOU
FUNCTION_BLOCK PUBLIC EventMsg
VAR_INPUT

END_VAR
VAR_OUTPUT
END_VAR
VAR
	CfgEvent                : TcEvent;
    fbEvent                 : ADSLOGEVENT;
    bSetEvent               : BOOL;(* Rising edge sets event *)  
	bInitialize : BOOL := TRUE;
END_VAR

IF (bInitialize) THEN
	CfgEvent.Class := TCEVENTCLASS_ALARM;
	CfgEvent.Prio := 2;
	CfgEvent.Id := 1;
	CfgEvent.SourceId := 17001;
	CfgEvent.bQuitRequired := FALSE;//TRUE;
	CfgEvent.Flags := TCEVENTFLAG_LOG OR TCEVENTFLAG_SRCID OR TCEVENTFLAG_AUTOFMTALL;
	CfgEvent.StreamType := TCEVENTSTREAM_SIMPLE;
	CfgEvent.ProgId :='TcEventFormatter.TcXMLFormatter' ;
    bInitialize:= FALSE;	
END_IF

fbEvent(Event:=FALSE);

METHOD PUBLIC SendEventMsg : BOOL
VAR_INPUT
	MsgClass :		UDINT;
	EventID :		UDINT;
	SourceID : 		UDINT;
END_VAR

CfgEvent.Class := MsgClass;
CfgEvent.Id := EventID;
CfgEvent.SourceId := SourceID;
fbEvent( NETID:= '',
        PORT:= 110,
        Event:=TRUE,					//Looking for rising edge here.
        EventConfigData:= CfgEvent,        
        TMOUT:= T#3S);
fbEvent(Event:= FALSE);		// transition, if not already done to falling edge
END_METHOD

END_FUNCTION_BLOCK

// ---- POUs/FrameworkPOUs/EventMsgParams.TcPOU
FUNCTION_BLOCK PUBLIC EventMsgParams
VAR_INPUT
	
END_VAR
VAR_OUTPUT
END_VAR
VAR
	CfgEvent                : TcEvent;
    fbEvent                 : ADSLOGEVENT;
    bSetEvent               : BOOL;(* Rising edge sets event *)
    eventData               : ST_EventData;
    TcEventDataFormatString : STRING    := '%f%d';
	bInitialize : BOOL := TRUE;
END_VAR

IF (bInitialize) THEN
	CfgEvent.Class := TCEVENTCLASS_ALARM;
	CfgEvent.Prio := 2;
	CfgEvent.Id := 1;
	CfgEvent.SourceId := 17001;
	CfgEvent.bQuitRequired := FALSE;//TRUE;
	CfgEvent.DataFormatStrAddress := ADR(TcEventDataFormatString);
	CfgEvent.Flags := TCEVENTFLAG_LOG OR TCEVENTFLAG_SRCID OR TCEVENTFLAG_AUTOFMTALL;
	CfgEvent.StreamType := TCEVENTSTREAM_SIMPLE;
	CfgEvent.ProgId :='TcEventFormatter.TcXMLFormatter' ;	
	eventData.rVal     := 0.00;
	eventData.iVal    := 0;
	bInitialize:= FALSE;	
END_IF

fbEvent(Event:=FALSE);

METHOD PUBLIC SendEventMsgParams : BOOL
VAR_INPUT
	MsgClass :		UDINT;
	EventID :		UDINT;
	SourceID : 		UDINT;
	RealVal: 		LREAL;
	IntVal :  		UDINT;
END_VAR
CfgEvent.Class := MsgClass;
CfgEvent.Id := EventID;
CfgEvent.SourceId := SourceID;
eventData.rVal := RealVal;
eventData.iVal := IntVal;
fbEvent( NETID:= '',
        PORT:= 110,
        Event:=TRUE,
        EventConfigData:= CfgEvent,
        EventDataAddress := ADR(eventData) ,
    	EventDataLength := SIZEOF(eventData),
        TMOUT:= T#3S);
END_METHOD

END_FUNCTION_BLOCK

// ---- POUs/MagneMotion/MMClient.TcPOU
FUNCTION_BLOCK PUBLIC MMClient
VAR_INPUT
	sSrvNetID	: T_AmsNetID	:= '';(* TwinCAT TCP/IP server network address *)
	sRemoteHost	: T_IPv4Addr 	:= '192.168.0.61';(* Server IP network address *)
	nRemotePort	: UDINT 		:= 799;(* Server port number *)
	bEnable		: BOOL 			:= TRUE;(* TRUE => enable client data exchange, FALSE => disable *)
	bLog		: BOOL 			:= FALSE;//TRUE;(* TRUE => Enable log message output, FALSE => Disable *)
	sPrefix		: STRING 		:= 'MM CLIENT::';(* Log message description string (allows the identification of log message source) *)
END_VAR
VAR_OUTPUT
	eState		: E_SocketConnectionState := eSOCKET_DISCONNECTED;(* TCP/IP connection state *)
END_VAR
VAR 
	fbConnection	: HLCConnection;(* Client data exchange control function block *)
	fbTx 			: FB_Tx_FrameFifo;(* Tx fifo *)
	fbRx 			: FB_Rx_FrameFifo;(* Rx fifo *)
	fbLog			: FB_LogFifo;(* Log/debug/error fifo *)
END_VAR

fbConnection( 	sSrvNetID := sSrvNetID, fbRx := fbRx, fbTx := fbTx, fbLog := fbLog, 
				bEnable := bEnable, sRemoteHost := sRemoteHost, nRemotePort := nRemotePort,  
				bLog := bLog, sPrefix := sPrefix, eState=>eState );

END_FUNCTION_BLOCK

// ---- POUs/MagneMotion/HLCConnection.TcPOU
(* This function block provides a socket and connection to the Magnemotion HLC *)
(* TxFifo is checked for any packets to send, if there are any, this fb will manage sending them *)
(* Any received data is properly checked for length and inserted into the RxFifo tail *)
FUNCTION_BLOCK PUBLIC HLCConnection
VAR_IN_OUT
	fbTx 		: FB_Tx_FrameFifo;(* TX fifo *)
	fbRx 		: FB_Rx_FrameFifo;(* RX fifo *)
	fbLog		: FB_LogFifo;(* Log message fifo *)
END_VAR

VAR_INPUT
	sSrvNetID	: T_AmsNetID	:= '';(* TwinCAT TCP/IP server network address *)
	sRemoteHost	: T_IPv4Addr 	:= '192.168.0.61';(* IP address of remote server *)
	nRemotePort	: UDINT			:= 799;(* Remote server port *)
	bEnable		: BOOL			:= FALSE;(* TRUE => Enable/connect, FALSE => Disable/disconnect *)
	tReconnect	: TIME 			:= T#10S;(* Try to reconnect after this time *)
	bLog		: BOOL 			:= FALSE; (* TRUE => Enable debug output, FALSE => Disable debug output *)
	sPrefix		: STRING 		:= 'CLIENT::';(* Log message description string (allows the identification of log message source) *)
END_VAR

VAR_OUTPUT
	eState		: E_SocketConnectionState := eSOCKET_DISCONNECTED;(* TCP/IP connection state *)
END_VAR

VAR
	fbConnect 	: FB_ClientServerConnection;(* Create/release TCP/IP connection *)
	fbSend		: FB_SocketSend;(* Send TCP/IP data *)
	fbReceive	: FB_SocketReceive;(* Receive TCP/IP data *)
	nState 		: BYTE;(* Global state *)
	bSndBusy 	: BOOL;(* Tx state *)
	bRcvBusy 	: BOOL;(* Rx state *)
	bDisconnect	: BOOL;(* Disconnect flag, if set the socket will be closed *)

	fbPollTimer	: TON;(* Rx data poll timer *)
	fbResponseTimer	: TON;(* Response timeout timer *)
	fbReconnectTimer : TON;(* Reconnect timer *)

	nS			: UDINT;(* Send frame counter *)
	nR			: UDINT;(* Received frame counter *)
	cbReceived	: UDINT;(* Count of received data bytes *)
	rxBuffer	: ARRAY[0..MM_CONST.PLCPRJ_BUFFER_SIZE] OF BYTE;
	cbFrame		: UDINT;(* Rx frame byte size *)
	stTxFrame	: ST_MM_TxFrame;(* Tx frame buffer (inclusive header) *)
	stRxFrame	: ST_MM_RxFrame;(* Rx frame buffer (inclusive header) *)
	bAbort		: BOOL;(* Flag to abort frame parsing loop *)
	event		: FB_SimpleAdsLogEvent;
	
	bInitialize : BOOL := TRUE;
	fbCloseAll		: FB_SocketCloseAll;
	
END_VAR

fbCloseAll( sSrvNetID := sSrvNetID, bExecute:= bInitialize );
IF fbCloseAll.bBusy OR fbCloseAll.bError THEN
	RETURN;
END_IF
bInitialize := FALSE;
CASE nState OF
	0:(* Create TCP/IP connection *)
		fbConnect( 	sSrvNetID 		:= sSrvNetID,
					nMode			:= SEL( bLog, 0, CONNECT_MODE_ENABLEDBG ),(* Enable/disable debug output *)
					sRemoteHost 	:= sRemoteHost,
					nRemotePort 	:= nRemotePort,
					tReconnect		:= tReconnect,
					bEnable			:= bEnable,
					eState			=> eState );
		IF NOT fbConnect.bBusy THEN
			IF NOT fbConnect.bError THEN
				IF eState = eSOCKET_CONNECTED THEN(* we are connected *)
					
					fbTx.Clear( sPrefix := CONCAT( sPrefix, 'FB_Tx_FrameFifo(sender)::' ), bLog := bLog );(* Clear TX fifo (optional) *)
					fbRx.Clear( sPrefix := CONCAT( sPrefix, 'FB_Rx_FrameFifo(receiver)::' ), bLog := bLog );(* Clear RX fifo (optional) *)
					fbLog.Clear( sPrefix := sPrefix, bLog := bLog );(* Clear log fifo (optional) *)
					bSndBusy := FALSE;
					bRcvBusy := FALSE;
					bDisconnect := FALSE;
					cbReceived 	:= 0;(* Reset number of received data bytes *)
					nR 			:= 0;(* Reset receive frame counter *)
					nS 			:= 0;(* Reset send frame counter *)

					fbPollTimer( IN := FALSE, PT := T#0S );
					fbResponseTimer( IN := FALSE, PT := MM_CONST.PLCPRJ_RECEIVE_TIMEOUT );
					fbReconnectTimer( IN := FALSE, PT := tReconnect );
				    //event(SourceID := 17001,EventID:=1,bSetEvent := TRUE, bQuit :=FALSE); 
					fbLog.Message( sMessage := 'Connection established!', hSocket := fbConnect.hSocket );
					nState 	:= 1;
				END_IF
			ELSE(* Connect error => log error *)
				fbLog.Error( sMessage := 'FB_ClientServerConnection()', nErrID := fbConnect.nErrId );
				 //event(SourceID := 17001,EventID:=1,bSetEvent := TRUE, bQuit :=FALSE); 
			END_IF
		END_IF


	1:(* Data exchange state *)
		bDisconnect := NOT bEnable OR bDisconnect;(* User/internal disconnect requested? *)
		IF bDisconnect AND NOT bSndBusy AND NOT bRcvBusy THEN
			bDisconnect := FALSE;
			fbLog.Message( sMessage := 'Closing connection!', hSocket := fbConnect.hSocket );
			nState := 2;(* Disconnect *)
		ELSE

			(* --------------------------- Send tx data --------------------------------- *)
			IF NOT bDisconnect AND NOT bSndBusy THEN
				fbTx.RemoveHead();(* Remove oldest user data entry *)
				IF fbTx.bOk THEN(* Success *)
						
					stTxFrame := fbTx.stGet;
					(* Properly formatted message is expected to be entered into the FIFO*)				
					(* Send frame *)
					fbSend( bExecute := FALSE );
					fbSend(	sSrvNetID 	:= sSrvNetID,
							hSocket		:= fbConnect.hSocket,
							cbLen		:= MM_CONST.TOTAL_MSG_LEN_ADJUST + stTxFrame.MsgLength,(* Size of header + size of user data *)
							pSrc		:= ADR(stTxFrame),(* Pointer to the frame data *)
							bExecute	:= TRUE );
					bSndBusy := TRUE;
				END_IF
			ELSE(* Wait until send not busy *)
				fbSend( bExecute := FALSE );
				IF NOT fbSend.bBusy THEN
					bSndBusy := FALSE;
					IF NOT fbSend.bError THEN(* No error *)
						nS := nS + 1;(* Increment the number of send frames *)
					ELSE(* Send error => Log error and disconnect *)
						fbLog.Error( sMessage := 'FB_SocketSend()', nErrID := fbSend.nErrId );
						bDisconnect := TRUE;(* Set flag *)
					END_IF
				END_IF
			END_IF
			(* -------------------------------------------------------------------------- *)

			(* ------------------ Get/fetch rx data ------------------------------------- *)
			IF NOT bDisconnect AND NOT bRcvBusy THEN
				fbPollTimer( IN := TRUE );
				IF fbPollTimer.Q THEN
					IF fbRx.cbFree >= SIZEOF(stRxFrame) THEN(* Check free rx fifo space *)
						fbPollTimer( IN := FALSE, PT := MM_CONST.PLCPRJ_RECEIVE_POLLING_TIME );
						fbReceive( bExecute := FALSE );
						fbReceive( 	sSrvNetId	:= sSrvNetID,
									hSocket		:= fbConnect.hSocket,
									cbLen		:= SIZEOF(rxBuffer) - cbReceived,
									pDest		:= ADR(rxBuffer) + cbReceived,
									bExecute	:= TRUE );
						bRcvBusy := TRUE;
					END_IF
				END_IF
				
			ELSE(* Wait until receive not busy *)
				
				fbReceive( bExecute := FALSE );
				IF NOT fbReceive.bBusy THEN
					bRcvBusy := FALSE;
					IF NOT fbReceive.bError THEN
						IF fbReceive.nRecBytes > 0 THEN (* Some bytes received *)

							fbPollTimer( IN := FALSE, PT := T#0S );(* Bytes received => increase the read (polling) speed *)
							fbResponseTimer( IN := FALSE );(* Bytes received => disable timeout check *)
							cbReceived := cbReceived + fbReceive.nRecBytes;

							(* Parse received bytes *)
							REPEAT
								bAbort := TRUE;(* Set flag *)
								
								IF (cbReceived >= MM_CONST.FRAMING_HEADER) THEN (* All header bytes received => check header data *)
									
									MEMCPY( ADR( stRxFrame ), ADR( rxBuffer ),MM_CONST.FRAMING_HEADER  );(* Get header data *)
								
									IF (stRxFrame.StartBytes = HOST_TO_BE16(16#ABBA)) (* Check start bytes *)
									AND (stRxFrame.MsgLength <= SIZEOF(stRxFrame))(* Check frame (user data) length *)
									THEN
									
										cbFrame := stRxFrame.MsgLength+MM_CONST.FRAMING_HEADER;(* Calculate the expected receive frame length *)
										IF cbReceived >= cbFrame  THEN (* All frame (user data) bytes received? *)
	
											MEMCPY( ADR( stRxFrame ), ADR( rxBuffer ), MIN( SIZEOF(stRxFrame), cbFrame ) );
											fbRx.AddTail( stPut := stRxFrame);(* Add user data to the rx fifo *)
											IF fbRx.bOk THEN
												nR := nR + 1;(* Increment receive counter *)

												MEMMOVE( ADR( rxBuffer ), ADR( rxBuffer ) + cbFrame, cbReceived - cbFrame );(* Shift the remaining rx bytes *)
												cbReceived := cbReceived - cbFrame;(* Recalculate the size of the remaining rx bytes *)

												IF fbRx.cbFree >= SIZEOF(stRxFrame) THEN
													bAbort := FALSE;(* reset flag, try to parse next frame *)
												END_IF
											ELSE (* Fifo overflow => log error and disconnect *)
												fbLog.Error( sMessage := 'FB_FrameFifo(receiver)', nErrID := MM_CONST.PLCPRJ_ERROR_RECFIFO_OVERFLOW );
												bDisconnect := TRUE;(* Set flag *)
												RETURN;
											END_IF

(*										ELSE repeat reading *)
										END_IF

									ELSE(* Receive error => Invalid frame format/data *)
										fbLog.Error( sMessage := 'FB_ClientConnection()', nErrID := MM_CONST.PLCPRJ_ERROR_INVALID_FRAME_FORMAT );
										bDisconnect := TRUE;(* Set flag *)
										RETURN;
									END_IF

(*								ELSE repeat reading *)
								END_IF (* IF cbReceived >= SIZEOF(stRxFrame.head) THEN *)

							UNTIL bAbort
							END_REPEAT

						ELSE(* No bytes received *)
							fbResponseTimer( IN := TRUE );(* No bytes received => enable timeout check *)
							IF fbResponseTimer.Q THEN (* Timeout error*)
								fbResponseTimer( IN := FALSE );
								fbLog.Error( sMessage := 'FB_ClientConnection()', nErrID := MM_CONST.PLCPRJ_ERROR_RECEIVE_TIMEOUT );
								bDisconnect := TRUE;(* Set flag *)
							END_IF							
						END_IF(* IF fbReceive.nRecBytes > 0 THEN *)

					ELSE(* Receive error => Log error and disconnect *)
						fbLog.Error( sMessage := 'FB_SocketReceive()', nErrID := fbReceive.nErrId );
						bDisconnect := TRUE;(* set flag *)
					END_IF

				END_IF(* IF NOT fbReceive.bBusy THEN *)
				
			END_IF(* IF NOT bDisconnect AND NOT bRcvBusy THEN *)
			(* -------------------------------------------------------------------------- *)
			
			
		END_IF(* IF bDisconnect AND NOT bSndBusy AND NOT bRcvBusy THEN *)


	2:(* Disconnect *)
		fbConnect( bEnable:= FALSE, eState=>eState );
		IF eState = eSOCKET_DISCONNECTED THEN
			fbReconnectTimer( IN := TRUE );(* Please wait some seconds and then try to connect again *)
			IF fbReconnectTimer.Q THEN
				fbReconnectTimer( IN := FALSE );
				//event(SourceID := 17001,EventID:=2,bSetEvent := TRUE, bQuit :=FALSE); 
				nState := 0;
			END_IF
		END_IF


END_CASE

END_FUNCTION_BLOCK

// ---- POUs/MagneMotion/HelperPOUs/FB_Tx_FrameFifo.TcPOU
(* Tx/Rx (string data) fifo control function block *)
FUNCTION_BLOCK FB_Tx_FrameFifo
VAR_INPUT
	bLog		: BOOL		:= FALSE;(* TRUE => Enable log message output, FALSE => Disable *)
	sPrefix		: STRING	:= 'Unknown::';(* Log message description string (allows the identification of log message source) *)
	stPut		: ST_MM_TxFrame;(* Frame to add (write) to the fifo *)
END_VAR
VAR_OUTPUT
	bOk			: BOOL; 	(* TRUE = New entry added or removed succesfully, FALSE = Fifo overflow or fifo empty *)
	stGet		: ST_MM_TxFrame;(* Frame removed (read) from fifo *)
	nCount		: UDINT		:= 0;(* Number of fifo entries *)
	cbFree		: UDINT 	:= 0;(* Free buffer space *)
END_VAR
VAR
	fbBuffer 	: FB_MemRingBuffer;(* Basic (lower level) buffer control function block *)
	buffer		: ARRAY[-3..MM_CONST.PLCPRJ_BUFFER_SIZE] OF BYTE;(* Internal buffer memory *)
END_VAR

;

ACTION AddTail:
(* Adds new fifo entry *)
fbBuffer.A_AddTail( pBuffer:= ADR(buffer), cbBuffer:= SIZEOF(buffer),
					pWrite := ADR( stPut ), cbWrite := SIZEOF( stPut ), 
					bOk=>bOk, nCount=>nCount );
IF bOk THEN
	cbFree := MM_CONST.PLCPRJ_BUFFER_SIZE - fbBuffer.cbSize;(* Calculate the free buffer space *)
	IF bLog THEN(* Log message *)
		F_ADSLOGHEXDATA( CONCAT( sPrefix, '<=' ), ADR( stPut ), SIZEOF( stPut ) );
	END_IF
END_IF
END_ACTION

ACTION Clear:
(* Resets fifo = clears all data *)
MEMSET( ADR( stGet ), 0, SIZEOF( stGet ) );
fbBuffer.A_Reset( pBuffer:= ADR(buffer), cbBuffer:= SIZEOF(buffer),
					pWrite := ADR( stPut ), cbWrite := SIZEOF( stPut ), 
					pRead := ADR( stGet ), cbRead := SIZEOF( stPut ),
					bOk=>bOk, nCount=>nCount );
cbFree := MM_CONST.PLCPRJ_BUFFER_SIZE;(* Free buffer size *)
END_ACTION

ACTION RemoveHead:
(* Removes oldest fifo entry *)
MEMSET( ADR( stGet ), 0, SIZEOF( stGet ) );
fbBuffer.A_RemoveHead( pBuffer:= ADR(buffer), cbBuffer:= SIZEOF(buffer),
						pRead := ADR( stGet ), cbRead := SIZEOF( stGet ),
						bOk=>bOk, nCount=>nCount );
IF bOk THEN
	cbFree := MM_CONST.PLCPRJ_BUFFER_SIZE - fbBuffer.cbSize;(* Calculate the free buffer space *)
END_IF
END_ACTION

END_FUNCTION_BLOCK

// ---- POUs/MagneMotion/HelperPOUs/F_ADSLOGHEXDATA.TcPOU
(* This function logs hexadecimal data to the TwinCAT XAE->Error list window *)
FUNCTION F_ADSLOGHEXDATA : DINT
VAR_INPUT
	sPrefix		: STRING;(* Debug message prefix string (allows the identification of log message source) *)
	pBuffer		: PVOID;(* Address of source buffer *)
	cbBuffer	: UDINT;(* Byte size of source buffer *)
END_VAR
VAR
	fbSplit	: FB_MemBufferSplit;
	sArg	: T_MaxString;
	sFormat : STRING;
END_VAR

IF pBuffer = 0 OR cbBuffer = 0 THEN
	RETURN;
END_IF

sFormat := CONCAT( sPrefix, '%s' );
fbSplit.eCmd := eEnumCmd_First;

REPEAT
	fbSplit( pBuffer := pBuffer, cbBuffer := cbBuffer, cbSize := 32 );(* Split binary data to 32 byte segments *)
	IF fbSplit.bOk THEN

		sArg := DATA_TO_HEXSTR( pData := fbSplit.pSegment, cbData := fbSplit.cbSegment, FALSE );(* Convert binary data to hex string *)

		F_ADSLOGHEXDATA := ADSLOGSTR( ADSLOG_MSGTYPE_HINT OR ADSLOG_MSGTYPE_LOG, sFormat, sArg );(* Log hex string *)

		sFormat := '%s';
		fbSplit.eCmd := eEnumCmd_Next;
	END_IF
UNTIL NOT fbSplit.bOk
END_REPEAT

END_FUNCTION

// ---- POUs/MagneMotion/HelperPOUs/FB_Rx_FrameFifo.TcPOU
(* Tx/Rx (string data) fifo control function block *)
FUNCTION_BLOCK FB_Rx_FrameFifo
VAR_INPUT
	bLog		: BOOL		:= FALSE;(* TRUE => Enable log message output, FALSE => Disable *)
	sPrefix		: STRING	:= 'Unknown::';(* Log message description string (allows the identification of log message source) *)
	stPut		: ST_MM_RxFrame;(* Frame to add (write) to the fifo *)
END_VAR
VAR_OUTPUT
	bOk			: BOOL; 	(* TRUE = New entry added or removed succesfully, FALSE = Fifo overflow or fifo empty *)
	stGet		: ST_MM_RxFrame;(* Frame removed (read) from fifo *)
	nCount		: UDINT		:= 0;(* Number of fifo entries *)
	cbFree		: UDINT 	:= 0;(* Free buffer space *)
END_VAR
VAR
	fbBuffer 	: FB_MemRingBuffer;(* Basic (lower level) buffer control function block *)
	buffer		: ARRAY[-3..MM_CONST.PLCPRJ_BUFFER_SIZE] OF BYTE;(* Internal buffer memory *)
END_VAR

;

ACTION AddTail:
(* Adds new fifo entry *)
fbBuffer.A_AddTail( pBuffer:= ADR(buffer), cbBuffer:= SIZEOF(buffer),
					pWrite := ADR( stPut ), cbWrite := SIZEOF( stPut ), 
					bOk=>bOk, nCount=>nCount );
IF bOk THEN
	cbFree := MM_CONST.PLCPRJ_BUFFER_SIZE - fbBuffer.cbSize;(* Calculate the free buffer space *)
	IF bLog THEN(* Log message *)
		F_ADSLOGHEXDATA( CONCAT( sPrefix, '<=' ), ADR( stPut ), SIZEOF( stPut ) );
	END_IF
END_IF
END_ACTION

ACTION Clear:
(* Resets fifo = clears all data *)
MEMSET( ADR( stGet ), 0, SIZEOF( stGet ) );
fbBuffer.A_Reset( pBuffer:= ADR(buffer), cbBuffer:= SIZEOF(buffer),
					pWrite := ADR( stPut ), cbWrite := SIZEOF( stPut ), 
					pRead := ADR( stGet ), cbRead := SIZEOF( stPut ),
					bOk=>bOk, nCount=>nCount );
cbFree := MM_CONST.PLCPRJ_BUFFER_SIZE;(* Free buffer size *)
END_ACTION

ACTION RemoveHead:
(* Removes oldest fifo entry *)
MEMSET( ADR( stGet ), 0, SIZEOF( stGet ) );
fbBuffer.A_RemoveHead( pBuffer:= ADR(buffer), cbBuffer:= SIZEOF(buffer),
						pRead := ADR( stGet ), cbRead := SIZEOF( stGet ),
						bOk=>bOk, nCount=>nCount );
IF bOk THEN
	cbFree := MM_CONST.PLCPRJ_BUFFER_SIZE - fbBuffer.cbSize;(* Calculate the free buffer space *)
END_IF
END_ACTION

END_FUNCTION_BLOCK

// ---- POUs/MagneMotion/HelperPOUs/FB_LogFifo.TcPOU
(* Log/debug/error message fifo *)
FUNCTION_BLOCK FB_LogFifo
VAR_INPUT
	bLog		: BOOL 		:= FALSE;(* TRUE => Enable log message output, FALSE => Disable *)
	sPrefix		: STRING 	:= 'Unknown::';(* Log message description string (allows the identification of log message source) *)
	
	sMessage	: STRING 	:= '';(* String message to add (write) to the fifo *)
	nErrID		: UDINT 	:= 0;(* Error code to add (write) to the fifo *)
	hSocket		: T_HSOCKET;(* Socket connection handle *)
END_VAR
VAR_OUTPUT
	bOk			: BOOL;(* TRUE = New entry added or removed succesfully, FALSE = Fifo overflow or fifo empty *)
	sGet		: T_MaxString := '';(* String entry removed (read) from fifo *)
	nCount		: UDINT := 0;(* Number of fifo entries *)
END_VAR
VAR
	fbBuffer 	: FB_StringRingBuffer;(* Basic (lower level) string buffer control function block *)
	buffer		: ARRAY[0..MM_CONST.PLCPRJ_BUFFER_SIZE] OF BYTE;(* Internal buffer memory *)
	sSource		: T_MaxString;	
	sPut		: T_MaxString;
END_VAR

;

ACTION Clear:
(* Clears all fifo entries *)
fbBuffer.A_Reset( 	pBuffer := ADR( buffer ), cbBuffer := SIZEOF( buffer ), 
					bOk=>bOk, nCount=>nCount, getValue=>sGet );
END_ACTION

ACTION Error:
(* Adds new fifo entry *)
IF nErrID = 0 THEN
	sSource := '::Error: 0x';
ELSIF ( nErrID AND 16#80000000) = 16#80000000 THEN
	IF nErrID = 16#80072746 THEN
		sSource := '::Win32 error (the connection is reset by remote side): 0x';
	ELSE
		sSource := '::Win32 error: 0x';
	END_IF
ELSIF (nErrID AND 16#00008100) = 16#00008100 THEN
	CASE nErrID OF
		MM_CONST.PLCPRJ_ERROR_RECEIVE_TIMEOUT:
			sSource := '::PLC sample project receive timeout error: 0x';
		MM_CONST.PLCPRJ_ERROR_SENDFIFO_OVERFLOW:
			sSource := '::PLC sample project send fifo overflow error: 0x';
		MM_CONST.PLCPRJ_ERROR_RECFIFO_OVERFLOW:
			sSource := '::PLC sample project receive fifo overflow error: 0x';
		MM_CONST.PLCPRJ_ERROR_INVALID_FRAME_FORMAT:
			sSource := '::PLC sample project invalid frame format error: 0x';
	ELSE
		sSource := '::Other PLC sample project error: 0x';
	END_CASE
ELSIF (nErrID AND 16#00008000) = 16#00008000 THEN
	sSource := '::Internal TCP/IP Connection Server error: 0x';
ELSE
	sSource := '::TwinCAT System error: 0x';
END_IF

sPut := CONCAT( CONCAT( CONCAT( sPrefix, sMessage ), sSource ), DWORD_TO_HEXSTR( nErrID AND 16#FFFF, 0, FALSE ) ); 

fbBuffer.A_AddTail( pBuffer:= ADR(buffer), cbBuffer:= SIZEOF(buffer),
					putValue:= sPut, bOk=>bOk, nCount=>nCount );
IF bOk THEN
	IF bLog THEN(* Log error message *)
		ADSLOGSTR( ADSLOG_MSGTYPE_ERROR OR ADSLOG_MSGTYPE_LOG, '%s', sPut );	
	END_IF
END_IF
END_ACTION

ACTION Message:
(* Adds new fifo entry *)
sPut := CONCAT( CONCAT( sPrefix, sMessage ), CONCAT( '::', HSOCKET_TO_STRING(hSocket) ) );
fbBuffer.A_AddTail( pBuffer:= ADR(buffer), cbBuffer:= SIZEOF(buffer),
					putValue:= sPut, bOk=>bOk, nCount=>nCount );
IF bOk THEN
	IF bLog THEN(* Log information message *)
		ADSLOGSTR( ADSLOG_MSGTYPE_HINT OR ADSLOG_MSGTYPE_LOG, '%s', sPut );	
	END_IF
END_IF
END_ACTION

ACTION Remove:
(* Removes oldest fifo entry *)
IF nCount = 0 THEN
	sGet := '';
	bOk := FALSE;
	RETURN;
END_IF

fbBuffer.A_RemoveHead( pBuffer:= ADR(buffer), cbBuffer:= SIZEOF(buffer),
						getValue=>sGet, bOk=>bOk, nCount=>nCount );
END_ACTION

END_FUNCTION_BLOCK

// ---- POUs/MagneMotion/MM_MsgFormatter.TcPOU
(* Implements the Magnemotion TCP/IP Protocol and adds to TxFifo*)
FUNCTION_BLOCK PUBLIC MM_MsgFormatter
VAR_IN_OUT
	fbTx 	:	FB_Tx_FrameFifo;
	fbLog	:	FB_LogFifo;
END_VAR
VAR_INPUT
END_VAR
VAR_OUTPUT
END_VAR
VAR
	stToServer		: ST_MM_TxFrame; (* Tx user data *)
	sLogMessage 	: T_MaxString := '';(* Log/debug/error message *)
	udiOrderNumb	: UDINT;
END_VAR

;

(* Request Status for HLC *)
METHOD PUBLIC M_CmdHLCStatus : BOOL
VAR_INPUT
END_VAR
VAR
	ID 		:UINT;
	CRC		:UINT;	
END_VAR
(* Request Status for HLC *)
	stToServer.StartBytes := HOST_TO_BE16(16#ABBA);
	stToServer.MsgLength  := MM_CONST.B5_CMD_LEN;
	stToServer.DataArray[0] := 16#B5;	
	stToServer.DataArray[1] := MM_CONST.STATUS_REQ_TYPE_HLC;
	ID := HOST_TO_BE16(16#0); (* can be omitted, but kept here for msg length*)	
	memcpy(ADR(stToServer.DataArray[2]), ADR(ID),SIZEOF(UINT));
    stToServer.DataArray[4]	:= 16#0; (* can be omitted, but kept here for msg length*)
	CRC := HOST_TO_BE16(F_DATA_TO_CRC16_CCITT(ADR(stToServer),MM_CONST.B5_CMD_LEN+MM_CONST.CRC_CALC_LEN_ADJUST,16#FFFF));
	memcpy(ADR(stToServer.DataArray[5]), ADR(CRC),SIZEOF(UINT));
 	fbTx.AddTail( stPut := stToServer );(* Put user data to the tx fifo *)
	IF NOT fbTx.bOk THEN(* Fifo overflow => Log error *)
		fbLog.Error( sMessage := 'FB_FrameFifo(sender)', nErrID := MM_CONST.PLCPRJ_ERROR_SENDFIFO_OVERFLOW );
	END_IF
END_METHOD

(* Reset Cmd for all paths *)
METHOD PUBLIC M_CmdResetPath : BOOL
VAR_INPUT
END_VAR
VAR
	PathID	:	UINT;
	CRC		:	UINT;	
END_VAR
(* Reset Cmd for all paths *)
	stToServer.StartBytes := HOST_TO_BE16(16#ABBA);
	stToServer.MsgLength  := MM_CONST.B8_CMD_LEN;	
	stToServer.DataArray[0] := 16#B8;	
	PathID		:= HOST_TO_BE16(0);		
	memcpy(ADR(stToServer.DataArray[1]), ADR(PathID),SIZEOF(UINT));    
	CRC := HOST_TO_BE16(F_DATA_TO_CRC16_CCITT(ADR(stToServer),MM_CONST.B8_CMD_LEN+MM_CONST.CRC_CALC_LEN_ADJUST,16#FFFF));
	memcpy(ADR(stToServer.DataArray[3]), ADR(CRC),SIZEOF(UINT));
	fbTx.AddTail( stPut := stToServer );(* Put user data to the tx fifo *)
	IF NOT fbTx.bOk THEN(* Fifo overflow => Log error *)
		fbLog.Error( sMessage := 'FB_FrameFifo(sender)', nErrID := MM_CONST.PLCPRJ_ERROR_SENDFIFO_OVERFLOW );
	END_IF
END_METHOD

METHOD PUBLIC M_CmdResumeMov : BOOL
VAR_INPUT
END_VAR
VAR
	PathID 		:UINT;
	CRC		:UINT;	
END_VAR
	stToServer.StartBytes := HOST_TO_BE16(16#ABBA);
	stToServer.MsgLength  := MM_CONST.B2_CMD_LEN;	
	stToServer.DataArray[0] := 16#B3;	
	PathID		:= HOST_TO_BE16(0);		
	memcpy(ADR(stToServer.DataArray[1]), ADR(PathID),SIZEOF(UINT));    
	CRC := HOST_TO_BE16(F_DATA_TO_CRC16_CCITT(ADR(stToServer),MM_CONST.B8_CMD_LEN+MM_CONST.CRC_CALC_LEN_ADJUST,16#FFFF));
	memcpy(ADR(stToServer.DataArray[3]), ADR(CRC),SIZEOF(UINT));
	fbTx.AddTail( stPut := stToServer );(* Put user data to the tx fifo *)
	IF NOT fbTx.bOk THEN(* Fifo overflow => Log error *)
		fbLog.Error( sMessage := 'FB_FrameFifo(sender)', nErrID := MM_CONST.PLCPRJ_ERROR_SENDFIFO_OVERFLOW );
	END_IF
END_METHOD

METHOD PUBLIC M_CmdStartupPath : BOOL
VAR_INPUT
END_VAR
VAR
	PathID 		:UINT;
	CRC		:UINT;	
END_VAR
	stToServer.StartBytes := HOST_TO_BE16(16#ABBA);
	stToServer.MsgLength  := MM_CONST.B2_CMD_LEN;	
	stToServer.DataArray[0] := 16#B2;	
	PathID		:= HOST_TO_BE16(0);		
	memcpy(ADR(stToServer.DataArray[1]), ADR(PathID),SIZEOF(UINT));    
	CRC := HOST_TO_BE16(F_DATA_TO_CRC16_CCITT(ADR(stToServer),MM_CONST.B8_CMD_LEN+MM_CONST.CRC_CALC_LEN_ADJUST,16#FFFF));
	memcpy(ADR(stToServer.DataArray[3]), ADR(CRC),SIZEOF(UINT));
	fbTx.AddTail( stPut := stToServer );(* Put user data to the tx fifo *)
	IF NOT fbTx.bOk THEN(* Fifo overflow => Log error *)
		fbLog.Error( sMessage := 'FB_FrameFifo(sender)', nErrID := MM_CONST.PLCPRJ_ERROR_SENDFIFO_OVERFLOW );
	END_IF
END_METHOD

METHOD PUBLIC M_CmdSuspendMov : BOOL
VAR_INPUT
END_VAR
VAR
	PathID 		:UINT;
	CRC		:UINT;	
END_VAR
	stToServer.StartBytes := HOST_TO_BE16(16#ABBA);
	stToServer.MsgLength  := MM_CONST.B2_CMD_LEN;	
	stToServer.DataArray[0] := 16#B4;	
	PathID		:= HOST_TO_BE16(0);		
	memcpy(ADR(stToServer.DataArray[1]), ADR(PathID),SIZEOF(UINT));    
	CRC := HOST_TO_BE16(F_DATA_TO_CRC16_CCITT(ADR(stToServer),MM_CONST.B8_CMD_LEN+MM_CONST.CRC_CALC_LEN_ADJUST,16#FFFF));
	memcpy(ADR(stToServer.DataArray[3]), ADR(CRC),SIZEOF(UINT));
	fbTx.AddTail( stPut := stToServer );(* Put user data to the tx fifo *)
	IF NOT fbTx.bOk THEN(* Fifo overflow => Log error *)
		fbLog.Error( sMessage := 'FB_FrameFifo(sender)', nErrID := MM_CONST.PLCPRJ_ERROR_SENDFIFO_OVERFLOW );
	END_IF
END_METHOD

(* Request Status for all Vehicles. This command will be called periodically by Monitoring loop *)
METHOD PUBLIC M_CmdVehicleStatus : BOOL
VAR_INPUT
END_VAR
VAR
	ID 		:UINT;
	CRC		:UINT;	
END_VAR
(* Request Status for Vehicle *)
	stToServer.StartBytes := HOST_TO_BE16(16#ABBA);
	stToServer.MsgLength  := MM_CONST.B5_CMD_LEN;
	stToServer.DataArray[0] := 16#B5;	
	stToServer.DataArray[1] := MM_CONST.STATUS_REQ_TYPE_Vehicle;
	ID := HOST_TO_BE16(16#0); (* can be omitted, but kept here for msg length*)	
	memcpy(ADR(stToServer.DataArray[2]), ADR(ID),SIZEOF(UINT));
    stToServer.DataArray[4]	:= 16#0; (* can be omitted, but kept here for msg length*)
	CRC := HOST_TO_BE16(F_DATA_TO_CRC16_CCITT(ADR(stToServer),MM_CONST.B5_CMD_LEN+MM_CONST.CRC_CALC_LEN_ADJUST,16#FFFF));
	memcpy(ADR(stToServer.DataArray[5]), ADR(CRC),SIZEOF(UINT));
 	fbTx.AddTail( stPut := stToServer );(* Put user data to the tx fifo *)
	IF NOT fbTx.bOk THEN(* Fifo overflow => Log error *)
		fbLog.Error( sMessage := 'FB_FrameFifo(sender)', nErrID := MM_CONST.PLCPRJ_ERROR_SENDFIFO_OVERFLOW );
	END_IF
END_METHOD

(* Add command to move vehicle to a position to the TxFifo with formatted expected by MM HLC*)
METHOD PUBLIC M_CmdVehToPos : BOOL
VAR_INPUT
	VehicleID 	: 	UINT;
	Flags 		: 	BYTE;
	Pos 		:	REAL;
	Acc			:	REAL;
	Vel			:	REAL;
END_VAR
VAR
	PathID 				:UINT;
	CRC					:UINT;
	OrderNumberLocal 	:UDINT;
	VehicleIDLocal		:UINT;	
    ConvertedDWord		:DWORD;
	FollowID			:UINT;
END_VAR
stToServer.StartBytes := HOST_TO_BE16(16#ABBA);
	stToServer.MsgLength  := MM_CONST.B1_CMD_LEN;	
	stToServer.DataArray[0] := 16#B1;
    IF (udiOrderNumb < 10000) THEN
		udiOrderNumb := udiOrderNumb+1;
	ELSE
        udiOrderNumb := 1;  			
	END_IF	
	OrderNumberLocal := HOST_TO_BE32(udiOrderNumb); //Local Copy
	memcpy(ADR(stToServer.DataArray[1]),ADR(OrderNumberLocal),SIZEOF(UDINT));
	VehicleIDLocal := HOST_TO_BE16(VehicleID);
	memcpy(ADR(stToServer.DataArray[5]),ADR(VehicleIDLocal),SIZEOF(UINT));
	memcpy(ADR(stToServer.DataArray[7]),ADR(Flags),SIZEOF(BYTE));
	
	memcpy(ADR(ConvertedDWord),ADR(Pos),SIZEOF(DWORD));
	
	memcpy(ADR(stToServer.DataArray[8]),ADR(ConvertedDWord),SIZEOF(DWORD));
	
	PathID		:= HOST_TO_BE16(1);		
	memcpy(ADR(stToServer.DataArray[12]), ADR(PathID),SIZEOF(UINT));

	memcpy(ADR(ConvertedDWord),ADR(Acc),SIZEOF(DWORD));
	
	memcpy(ADR(stToServer.DataArray[14]),ADR(ConvertedDWord),SIZEOF(DWORD));
	
	memcpy(ADR(ConvertedDWord),ADR(Vel),SIZEOF(DWORD));
	
	memcpy(ADR(stToServer.DataArray[18]),ADR(ConvertedDWord),SIZEOF(DWORD));
	
	FollowID := HOST_TO_BE16(0);
	memcpy(ADR(stToServer.DataArray[22]),ADR(FollowID),SIZEOF(DWORD));
	CRC := HOST_TO_BE16(F_DATA_TO_CRC16_CCITT(ADR(stToServer),MM_CONST.B1_CMD_LEN+MM_CONST.CRC_CALC_LEN_ADJUST,16#FFFF));
	memcpy(ADR(stToServer.DataArray[24]), ADR(CRC),SIZEOF(UINT));
	fbTx.AddTail( stPut := stToServer );(* Put user data to the tx fifo *)
	IF NOT fbTx.bOk THEN(* Fifo overflow => Log error *)
		fbLog.Error( sMessage := 'FB_FrameFifo(sender)', nErrID := MM_CONST.PLCPRJ_ERROR_SENDFIFO_OVERFLOW );
	END_IF
END_METHOD

END_FUNCTION_BLOCK

// ---- POUs/MagneMotion/MM_MsgParser.TcPOU
(* Implements the Magnemotion TCP/IP Protocol and adds to TxFifo*)
FUNCTION_BLOCK PUBLIC MM_MsgParser
VAR_IN_OUT
	fbRx : FB_Rx_FrameFifo;
	fbLog	:	FB_LogFifo;	
END_VAR
VAR_INPUT
END_VAR
VAR_OUTPUT
END_VAR
VAR
	stFromServer	: ST_MM_RxFrame; (* Rx user data *)
	sLogMessage 	: T_MaxString := '';(* Log/debug/error message *)
END_VAR

(*------------------------ Fetch rx data -------------------------------------- *)
REPEAT
	fbRx.RemoveHead( );(* fetch data from rx fifo *)
	IF fbRx.bOk THEN(* success *)

		(* TODO: Implement receive handler *)
		stFromServer := fbRx.stGet; 
		M_ResHLCMsg();

	END_IF
UNTIL NOT fbRx.bOk
END_REPEAT

(*---------------------- Get log/error messages from log fifo ------------------*)
REPEAT
	fbLog.Remove( );
	IF fbLog.bOk THEN

		(* TODO: Implement log message handler *)
		sLogMessage := fbLog.sGet;

	END_IF
UNTIL NOT fbLog.bOk
END_REPEAT

METHOD PUBLIC M_ResD0_B1Cmd : BOOL
VAR_INPUT
END_VAR
VAR
	LocalOrderNumb :DWORD;
	LocalOrderNumbBE: DWORD;
	LocalVehicleID : UINT;
	LocalVehicleIDBE: UINT;
END_VAR
memcpy(ADR(LocalOrderNumbBE),ADR(stFromServer.Resdata.DataArray[2]),SIZEOF(DWORD));
LocalOrderNumb := BE32_TO_HOST(LocalOrderNumbBE);
memcpy(ADR(LocalVehicleIDBE),ADR(stFromServer.Resdata.DataArray[6]),SIZEOF(UINT));
LocalVehicleID := BE16_TO_HOST(LocalVehicleIDBE);
IF (stFromServer.Resdata.ResCmdData.D0Res.CmdStatus = 16#00) THEN			
 	Stations.fbVehicleManager[LocalVehicleID].MoveCmdAccepted := TRUE; 
	ELSIF (stFromServer.Resdata.ResCmdData.D0Res.CmdStatus = 16#80) THEN 
		Stations.fbVehicleManager[LocalVehicleID].MoveCmdCmpl := TRUE; 
	ELSE			
		//Stations.VehicleManager[LocalVehicleID].VehMovePosState := eMM_VehMoveToPosCmdStatus.eMM_VehMoveToPosCmdRejected;
	END_IF
END_METHOD

METHOD PUBLIC M_ResD0_B2Cmd : BOOL
VAR_INPUT
END_VAR
IF (stFromServer.Resdata.ResCmdData.D0Res.CmdStatus = 16#00) THEN
	Stations.fbPrimeMover.StartupCmdState := eMM_StartupCmdStatus.eMM_StartupCmdAck;
ELSIF (stFromServer.Resdata.ResCmdData.D0Res.CmdStatus = 16#80) THEN
	Stations.fbPrimeMover.StartupCmdState := eMM_StartupCmdStatus.eMM_StartupCmdComplete;		
ELSE
	Stations.fbPrimeMover.StartupCmdState := eMM_StartupCmdStatus.eMM_StartupCmdRejected;
END_IF
END_METHOD

METHOD PUBLIC M_ResD0_B8Cmd : BOOL
VAR_INPUT
END_VAR
IF (stFromServer.Resdata.ResCmdData.D0Res.CmdStatus = 16#00) THEN
	Stations.fbPrimeMover.ResetCmdState := eMM_ResetCmdStatus.eMM_ResetCmdAck;
ELSIF (stFromServer.Resdata.ResCmdData.D0Res.CmdStatus = 16#80) THEN
	Stations.fbPrimeMover.ResetCmdState := eMM_ResetCmdStatus.eMM_ResetCmdComplete;
ELSE
	Stations.fbPrimeMover.ResetCmdState := eMM_ResetCmdStatus.eMM_ResetCmdRejected;
END_IF
END_METHOD

METHOD PUBLIC M_ResD1_HLCStatus : BOOL
VAR_INPUT
END_VAR
CASE stFromServer.Resdata.ResCmdData.D1Res.HLC_State OF
			MM_CONST.HLC_STATE_INIT:		
				Stations.fbPrimeMover.HLCState := eMM_HLCStatus.eHLC_STATE_INIT;	
			MM_CONST.HLC_STATE_DEGRADED:
                Stations.fbPrimeMover.HLCState := eMM_HLCStatus.eHLC_STATE_DEGRADED;			
		    MM_CONST.HLC_STATE_OPERATIONAL:
				Stations.fbPrimeMover.HLCState := eMM_HLCStatus.eHLC_STATE_OPERATIONAL;
			ELSE
				Stations.fbPrimeMover.HLCState := eMM_HLCStatus.eHLC_STATE_DEGRADED;						
		END_CASE
END_METHOD

METHOD PUBLIC M_ResD5_VehStatus : BOOL
VAR_INPUT
END_VAR
VAR
	LocalOrderNumb :DWORD;
	LocalOrderNumbBE: DWORD;
	LocalVehicleID : UINT;
	LocalVehicleIDBE: UINT;
	LocalPathIDBE: UINT;
	LocalPathID :UINT;
	LocalDestPathIDBE: UINT;
	LocalDestPathID :UINT;
	LocalVehPos: REAL;
	LocalVehVel:REAL;
	LocalVehCmdPos :REAL;
END_VAR
//VehicleID
memcpy(ADR(LocalVehicleIDBE),ADR(stFromServer.Resdata.DataArray[0]),SIZEOF(UINT));
LocalVehicleID := BE16_TO_HOST(LocalVehicleIDBE);
Status.MMVehiclesStatus[LocalVehicleID].VehicleID := LocalVehicleID; 

//Vehicle Present
Status.MMVehiclesStatus[LocalVehicleID].VehiclePresent := stFromServer.Resdata.DataArray[2]; 

//Path ID
memcpy(ADR(LocalPathIDBE),ADR(stFromServer.Resdata.DataArray[3]),SIZEOF(UINT));
LocalPathID := BE16_TO_HOST(LocalPathIDBE);
Status.MMVehiclesStatus[LocalVehicleID].PathID := LocalPathID; 

//DestinationPathID
memcpy(ADR(LocalDestPathIDBE),ADR(stFromServer.Resdata.DataArray[5]),SIZEOF(UINT));
LocalDestPathID := BE16_TO_HOST(LocalDestPathIDBE);
Status.MMVehiclesStatus[LocalVehicleID].DestinationPathID := LocalDestPathID; 

//VehiclePos
memcpy(ADR(LocalVehPos),ADR(stFromServer.Resdata.DataArray[7]),SIZEOF(DWORD));
Status.MMVehiclesStatus[LocalVehicleID].VehiclePos := LocalVehPos; 

//VehicleVel
memcpy(ADR(LocalVehVel),ADR(stFromServer.Resdata.DataArray[11]),SIZEOF(DWORD));
Status.MMVehiclesStatus[LocalVehicleID].Velocity := LocalVehVel; 

//VehicleCmdType
Status.MMVehiclesStatus[LocalVehicleID].VehicleCmdType := stFromServer.Resdata.DataArray[15]; 

//Vehicle Flags
Status.MMVehiclesStatus[LocalVehicleID].VehicleFlags := stFromServer.Resdata.DataArray[16]; 

// VehicleCmdPos
memcpy(ADR(LocalVehCmdPos),ADR(stFromServer.Resdata.DataArray[17]),SIZEOF(DWORD));
Status.MMVehiclesStatus[LocalVehicleID].VehicleCmdPos := LocalVehCmdPos; 

(* Copy Status into Byte Array for ADS Communication with HMI *) 
  
  (****************************************
	VehicleID			:	UINT; // 2 bytes
	VehiclePresent		:	BYTE; // 1 byte 
	PathID				:	UINT; // 2 bytes 
	DestinationPathID	:	UINT; // 2 bytes
	VehiclePos			: 	REAL; // 4 bytes
	Velocity			: 	REAL; // 4 bytes 
	VehicleCmdType		: 	BYTE; // 1 byte
	VehicleFlags		: 	BYTE; // 1 byte
	VehicleCmdPos		: 	REAL; // 4 bytes
	*****************************************)
(*
memset(ADR(Status.MMVehiclesStatusHMI[LocalVehicleID].VehicleStatusBytes), 0, SIZEOF (ST_VehicleStatusHMI.VehicleStatusBytes));
memcpy(ADR(Status.MMVehiclesStatusHMI[LocalVehicleID].VehicleStatusBytes[0]),ADR(LocalVehicleID),SIZEOF(UINT));
memcpy(ADR(Status.MMVehiclesStatusHMI[LocalVehicleID].VehicleStatusBytes[2]),ADR(Status.MMVehiclesStatus[LocalVehicleID].VehiclePresent),SIZEOF(BYTE));
memcpy(ADR(Status.MMVehiclesStatusHMI[LocalVehicleID].VehicleStatusBytes[3]),ADR(LocalPathID),SIZEOF(UINT));	
memcpy(ADR(Status.MMVehiclesStatusHMI[LocalVehicleID].VehicleStatusBytes[5]),ADR(LocalDestPathID),SIZEOF(UINT));
memcpy(ADR(Status.MMVehiclesStatusHMI[LocalVehicleID].VehicleStatusBytes[7]),ADR(LocalVehPos),SIZEOF(REAL));
memcpy(ADR(Status.MMVehiclesStatusHMI[LocalVehicleID].VehicleStatusBytes[11]),ADR(LocalVehVel),SIZEOF(REAL));
memcpy(ADR(Status.MMVehiclesStatusHMI[LocalVehicleID].VehicleStatusBytes[15]),ADR(Status.MMVehiclesStatus[LocalVehicleID].VehicleCmdType),SIZEOF(BYTE));
memcpy(ADR(Status.MMVehiclesStatusHMI[LocalVehicleID].VehicleStatusBytes[16]),ADR(Status.MMVehiclesStatus[LocalVehicleID].VehicleFlags),SIZEOF(BYTE));
memcpy(ADR(Status.MMVehiclesStatusHMI[LocalVehicleID].VehicleStatusBytes[17]),ADR(LocalVehCmdPos),SIZEOF(DWORD));
*)
(* End Copy for HMI ADS Communication*)
END_METHOD

METHOD PUBLIC M_ResHLCMsg : BOOL
VAR_INPUT
END_VAR
CASE (stFromServer.ResHeader) OF
16#D0:	
	CASE (stFromServer.Resdata.ResCmdData.D0Res.Cmd) OF
		16#B1:
			M_ResD0_B1Cmd();
		16#B2:
		    M_ResD0_B2Cmd();
		16#B3:
		16#B4:
		16#B5:
		16#B8:
		     M_ResD0_B8Cmd();			
	END_CASE
16#D1:
		M_ResD1_HLCStatus();
16#D2:
16#D3:
16#D4:
16#D5:
      M_ResD5_VehStatus();
16#D7:
ELSE	
//	Reset();
END_CASE
END_METHOD

END_FUNCTION_BLOCK

// ---- POUs/MagneMotion/MMStatusMonitor.TcPOU
FUNCTION_BLOCK PUBLIC MMStatusMonitor
VAR_IN_OUT
	
END_VAR
VAR_INPUT
END_VAR
VAR_OUTPUT
END_VAR
VAR
	HLCStatusTimer		:TON;
	PathStatusTimer		:TON;
	MotorStatusTimer	:TON;
	VehicleStatusTimer	:TON;
	byCounter: BYTE := 1;
	bVehicleJammed: BOOL := FALSE;
	bVehicleLostByMotor: BOOL := FALSE;
	bPrevVehicleJammed : BOOL := FALSE;
	JamTimer :TON;
END_VAR

HLCStatusTimer(IN:=TRUE,PT:=MM_CONST.MM_HLC_STATUS_POLLING);
PathStatusTimer(IN:=TRUE,PT:=MM_CONST.MM_PATH_STATUS_POLLING);
MotorStatusTimer(IN:=TRUE,PT:=MM_CONST.MM_MOTOR_STATUS_POLLING);
VehicleStatusTimer(IN:=TRUE, PT:=MM_CONST.MM_VEHICLE_STATUS_POLLING);

IF (HLCStatusTimer.Q) THEN
		Stations.fbMMSendMsg.M_CmdHLCStatus();
		HLCStatusTimer(IN:=FALSE);
END_IF

IF (PathStatusTimer.Q) THEN
		Stations.fbMMSendMsg.M_CmdHLCStatus(); // to do get path status
		PathStatusTimer(IN:=FALSE);
END_IF

IF (MotorStatusTimer.Q) THEN
		Stations.fbMMSendMsg.M_CmdHLCStatus(); // to do get HLC Status
		MotorStatusTimer(IN:=FALSE);
END_IF

IF (VehicleStatusTimer.Q) THEN
		Stations.fbMMSendMsg.M_CmdVehicleStatus();
		VehicleStatusTimer(IN:=FALSE);
END_IF

bVehicleJammed := FALSE;
bVehicleLostByMotor := FALSE;
FOR byCounter := 1 TO MM_CONST.MAX_VEHICLES BY 1 DO
	bVehicleJammed := bVehicleJammed OR STATUS.MMVehiclesStatus[byCounter].VehicleFlags.2;
	bVehicleLostByMotor := bVehicleLostByMotor OR (STATUS.MMVehiclesStatus[byCounter].VehicleFlags.0 = 0) OR (STATUS.MMVehiclesStatus[byCounter].VehicleFlags.7 = 1);
    STATUS.PartStatusHMI[byCounter] := PartsData.Status[byCounter].OverallStatus;	// this will add color to the vehicles on the HMI
	IF (STATUS.MMVehiclesStatus[byCounter].VehicleFlags.2) THEN STATUS.PartStatusHMI[byCounter] := ePartStatus.eJam; END_IF
END_FOR

IF (bVehicleJammed AND NOT bPrevVehicleJammed) THEN // only when transitioning from non-jammed state to jammed state
	//Stations.fbMMSendMsg.M_CmdSuspendMov();
	//GVL_IO.MM_YEnableMagneMotion := FALSE;
END_IF
bPrevVehicleJammed := bVehicleJammed;  // to ensure that after turning on the MM bus, we don't immediately shut down the MM bus.

IF (bVehicleJammed) THEN JamTimer(IN:=TRUE, PT:=T#40S);
	ELSE 
	JamTimer(IN:=FALSE);
END_IF
IF (GVL_IO.ResumeMovementFromHMI <>0) THEN // Button Click Resume From HMI.
//	Stations.fbMMSendMsg.M_CmdResumeMov();
	GVL_IO.ResumeMovementFromHMI := 0;
	GVL_IO.MM_YEnableMagneMotion := TRUE;
	Stations.fbPrimeMover.ResetPrimeMoverAndPurge(); // this will send prime mover to purrge state
	Stations.fbCycleControl.ResetCycleControlState();

	Stations.fbLoad1Sta.ClearVehicleTrigger();
	Stations.fbLoad2Sta.ClearVehicleTrigger(); 
	Stations.fbLoad3Sta.ClearVehicleTrigger();
	Stations.fbLoad4Sta.ClearVehicleTrigger();
	Stations.fbVisionSta.ClearVehicleTrigger();
	Stations.fbPistonSta.ClearVehicleTrigger();
	Stations.fbCapInsertSta.ClearVehicleTrigger();
	//Stations.fbGoodUnloadSta.ClearVehicleTrigger();
	Stations.fbGoodULSta_1.ClearVehicleTrigger();
	Stations.fbGoodULSta_2.ClearVehicleTrigger();
	Stations.fbGoodULSta_3.ClearVehicleTrigger();
	Stations.fbGoodULSta_4.ClearVehicleTrigger();
	Stations.fbRejectSta.ClearVehicleTrigger();
	Stations.fbIB_StopRobotSta.ClearVehicleTrigger();	
	Stations.fbOB_StopBeforeVisionSta.ClearVehicleTrigger(); 
	Stations.fbOB_StopRobotSta.ClearVehicleTrigger();
	Stations.fbOB_StopRobotSta.MoveToLoading := TRUE;
	
	Stations.fbRoutePlanner.SetRejectLoadPosChoiceToInit();
	Stations.fbRoutePlanner.SetGoodULLoadPosChoiceToInit();
	
	FOR byCounter := 1 TO MM_CONST.MAX_VEHICLES BY 1 DO
			Stations.fbVehicleManager[byCounter].ResetVehicleManager();
	END_FOR	
	
	IF (bVehicleLostByMotor) THEN
		;
	END_IF
END_IF

PROPERTY PUBLIC IsMMJammed : BOOL
GET
IsMMJammed := (JamTimer.Q);
END_GET
SET
END_SET
END_PROPERTY

END_FUNCTION_BLOCK

// ---- POUs/CycleControl.TcPOU
FUNCTION_BLOCK PUBLIC CycleControl
VAR_IN_OUT
	
END_VAR
VAR_INPUT
END_VAR
VAR_OUTPUT
END_VAR
VAR
	bInitialize : BOOL := TRUE;
	bFirst: BOOL := TRUE;
	State : eCycleControlState := eCycleControlState.eUnknown;
	NextState : eCycleControlState := eCycleControlState.eUnknown;
	byCounter: BYTE :=1;
	StateTimer : TON;
	//fbPID: FB_CTRL_PID;
	CycleStopReq : BOOL := FALSE;
END_VAR

IF (bInitialize) THEN
	bInitialize := FALSE;
	// to add all initialization code here
END_IF


CASE State OF
eCycleControlState.eUnknown:
	IF (GVL_IO.MC_XStartPB AND GVL_IO.MC_XAirPressureOK AND GVL_IO.MC_NotEStopped) THEN // wait for start button when powered up or PLC program restarted
		NextState := eCycleControlState.eInit;	   
	END_IF
    StackLightRed();
	
	StateTimer(IN:=TRUE, PT:= T#10S); // give a message out every 10 seconds
	IF (StateTimer.Q) THEN
		Logging.fbEventMsg.SendEventMsg(MsgClass := TCEVENTCLASS_STATEINFO, EventID:= Logging.ID_CY_Unknown, SourceID:= Logging.SrcCyclePOU);
		StateTimer(IN:=FALSE);
	END_IF

eCycleControlState.eInit:
	IF (Stations.fbPrimeMover.WaitingForHomingTrigger) THEN  // checking to see if Magnemotion has completed software Path reset and HLC operational
		NextState := eCycleControlState.eWaitForHoming;
	END_IF
	StateTimer(IN:=TRUE, PT := T#250MS);
	IF (StateTimer.Q) THEN
		GVL_IO.MC_YStackLightRed := NOT GVL_IO.MC_YStackLightRed;
		GVL_IO.MC_YStackLightYellow := NOT GVL_IO.MC_YStackLightYellow;
		GVL_IO.MC_YStackLightGreen := NOT GVL_IO.MC_YStackLightGreen;
		StateTimer(IN:=FALSE);
	END_IF
	

eCycleControlState.eWaitForHoming:
	(*IF(Stations.fbPistonSta.Ready AND Stations.fbCapInsertSta.Ready AND Stations.fbGoodUnloadSta.Ready AND Stations.fbRejectSta.Ready) THEN
		NextState := eCycleControlState.eReady;
	END_IF *)
	StackLightYellow();
	IF(Stations.fbLoad1Sta.Ready AND
       Stations.fbVisionSta.Ready AND  
       Stations.fbPistonSta.Ready AND 
       Stations.fbCapInsertSta.Ready AND 
       //Stations.fbGoodUnloadSta.Ready AND
       Stations.fbGoodULSta_1.Ready AND
		Stations.fbGoodULSta_2.Ready AND
		Stations.fbGoodULSta_3.Ready AND
		Stations.fbGoodULSta_4.Ready AND     
		Stations.fbAutoBagger.Ready AND     
	   Stations.fbRejectSta.Ready  
       ) THEN
		NextState := eCycleControlState.eReady;
		StackLightGreen();
		Stations.fbPrimeMover.TriggerAction := TRUE; // Enable the Magnemotion controller bus propulsion
	END_IF

eCycleControlState.eReady:
	//IF (GVL_IO.MC_XStartPB) THEN //need to change this later
		NextState := eCycleControlState.eAutoRun;   //don't really need this start button again 			
	//END_IF	

eCycleControlState.eAutoRun:
	IF(bFirst) THEN
		FOR byCounter := 1 TO MM_CONST.MAX_VEHICLES BY 1 DO
			Stations.fbVehicleManager[byCounter].M_SetNextMoveParams(MM_CONST.REJECT_ULOAD_POS,2.0,2.0,MM_CONST.REJECT_ULOAD_STA);
			Stations.fbVehicleManager[byCounter].TriggerVehMov := TRUE;			
		END_FOR	
	END_IF
	// to do add logic here to handle cycle stop
	NextState := eCycleControlState.eStartStop ;

eCycleControlState.eStartStop:	
	IF( Stations.fbMMMonitor.IsMMJammed OR 
		Stations.fbLoad1Sta.IsFaulted() OR 
		NOT Stations.fbBurnOffSta.IsAtTemperature OR 
		Stations.fbVisionSta.IsFaulted() OR 
        Stations.fbPistonSta.IsFaulted() OR 
       Stations.fbCapInsertSta.IsFaulted() OR 
       //Stations.fbGoodUnloadSta.IsFaulted() OR
		Stations.fbGoodULSta_1.IsFaulted() OR
		Stations.fbGoodULSta_2.IsFaulted() OR
		Stations.fbGoodULSta_3.IsFaulted() OR
		Stations.fbGoodULSta_4.IsFaulted() OR
		Stations.fbAutoBagger.IsFaulted() OR		            
        Stations.fbRejectSta.IsFaulted()) 
       THEN 
			StackLightRed();
			GVL_IO.YU_YIMBADIsOK := FALSE;
	END_IF
	
    IF( NOT Stations.fbMMMonitor.IsMMJammed AND
		NOT Stations.fbLoad1Sta.IsFaulted() AND 
	    Stations.fbBurnOffSta.IsAtTemperature AND 
	    NOT Stations.fbVisionSta.IsFaulted() AND 
        NOT Stations.fbPistonSta.IsFaulted() AND 
        NOT Stations.fbCapInsertSta.IsFaulted() AND 
        //NOT Stations.fbGoodUnloadSta.IsFaulted() AND
        NOT Stations.fbGoodULSta_1.IsFaulted() AND
		NOT Stations.fbGoodULSta_2.IsFaulted() AND
		NOT Stations.fbGoodULSta_3.IsFaulted() AND
		NOT Stations.fbGoodULSta_4.IsFaulted() AND   
		NOT Stations.fbAutoBagger.IsFaulted() AND
        NOT Stations.fbRejectSta.IsFaulted()) 
    THEN 
			StackLightGreen(); 
			GVL_IO.YU_YIMBADIsOK := TRUE;
	END_IF
    
    IF (NOT GVL_IO.MC_XStopPB) THEN // hit the stop button
		CycleStopReq := TRUE;		
	END_IF
	
    IF (GVL_IO.MC_XStopPB AND GVL_IO.MC_XStartPB) THEN 
		CycleStopReq := FALSE;		
	END_IF
    
   IF (GVL_IO.MachineEStopped OR NOT GVL_IO.MC_XAirPressureOK ) THEN 
		NextState := eCycleControlState.eWaitForHomingAfterEStop;
		StackLightRed();
    END_IF
	
	IF CycleStopReq THEN
		StackLightYellow(); // we have a stop request
	END_IF
	
	
eCycleControlState.eWaitForHomingAfterEStop:

	IF (GVL_IO.MC_XAirPressureOK AND GVL_IO.MC_NotEStopped) THEN // wait for start button when powered up or PLC program restarted
		IF(Stations.fbPistonSta.Ready AND Stations.fbCapInsertSta.Ready
        //AND Stations.fbGoodUnloadSta.Ready
        AND Stations.fbGoodULSta_1.Ready
		AND Stations.fbGoodULSta_2.Ready
		AND Stations.fbGoodULSta_3.Ready
		AND Stations.fbGoodULSta_4.Ready 
        AND Stations.fbVisionSta.Ready ) THEN // Maybe add other stations here as well
			NextState := eCycleControlState.eStartStop;
			StackLightGreen();
		END_IF
		IF (GVL_IO.MC_XStopPB AND GVL_IO.MC_XStartPB) THEN
			CycleStopReq := FALSE;
			///Stations.fbMMSendMsg.M_CmdResumeMov(); // allow accepting commands for vehicle movement ?? Need to try this
		END_IF		
	END_IF
	
	
eCycleControlState.eError:	
//fbPID;

IF (GVL_IO.MC_XStartPB) THEN 
	GVL_IO.MC_YStackLightYellow := TRUE;
END_IF

END_CASE

IF (State <> NextState) THEN
	bFirst := TRUE;
	StateTimer(IN:=FALSE);
ELSE 
	bFirst := FALSE;	
END_IF

State := NextState;
Status.StationsState[MM_CONST.CYCLE_CONTROL_HMI_STATE] := State;
AssignStationStatusForHMI();
AssignErrorMessagetoHMI();

PROPERTY AllowPrimeMoverEnable : BOOL
GET
AllowPrimeMoverEnable := (State = eCycleControlState.eStartStop);
END_GET
END_PROPERTY

METHOD PUBLIC AssignErrorMessagetoHMI : BOOL
VAR_INPUT
END_VAR
IF (Stations.fbMMMonitor.IsMMJammed) THEN
	Status.ErrorMessage := Status.PrimeMoverStatusMsg;
ELSIF (Stations.fbLoad1Sta.IsFaulted()) THEN
	Status.ErrorMessage := Status.Load1StatusMsg;
ELSIF(Stations.fbVisionSta.IsFaulted()) THEN
	Status.ErrorMessage := Status.VisionStatusMsg;
ELSIF(Stations.fbPistonSta.IsFaulted()) THEN
	Status.ErrorMessage := Status.PistonStatusMsg;
ELSIF(Stations.fbCapInsertSta.IsFaulted()) THEN
	Status.ErrorMessage := Status.CapStatusMsg; 
//ELSIF(Stations.fbGoodUnloadSta.IsFaulted()) THEN
//	Status.ErrorMessage := Status.GoodULStatusMsg;    
ELSIF(Stations.fbGoodULSta_1.IsFaulted()) THEN
	Status.ErrorMessage := Status.GoodUL_1_StatusMsg;       
ELSIF(Stations.fbGoodULSta_2.IsFaulted()) THEN
	Status.ErrorMessage := Status.GoodUL_2_StatusMsg;
ELSIF(Stations.fbGoodULSta_3.IsFaulted()) THEN
	Status.ErrorMessage := Status.GoodUL_3_StatusMsg;
ELSIF(Stations.fbGoodULSta_4.IsFaulted()) THEN
	Status.ErrorMessage := Status.GoodUL_4_StatusMsg;
ELSIF(Stations.fbRejectSta.IsFaulted()) THEN
	Status.ErrorMessage := Status.RejectStatusMsg;
ELSIF(Stations.fbAutoBagger.IsFaulted()) THEN
	Status.ErrorMessage := Status.AutoBaggerStatusMsg;
ELSIF (Stations.fbLoad1Sta.IsLoadWaitingForYushin()) THEN
	Status.ErrorMessage := Status.Load1StatusMsg;	
ELSE
	Status.ErrorMessage := '';
END_IF
END_METHOD

METHOD PUBLIC AssignStationStatusForHMI : BOOL
VAR_INPUT
END_VAR
Status.StationsState[MM_CONST.CYCLE_CONTROL_HMI_STATE] := State;

CASE State OF 
	eCycleControlState.eUnknown, eCycleControlState.eError:
		Status.StationStauts[MM_CONST.CYCLE_CONTROL_HMI_STATE] := OverallStationStatus.eError;
    eCycleControlState.eInit,eCycleControlState.eWaitForHoming:
	    Status.StationStauts[MM_CONST.CYCLE_CONTROL_HMI_STATE] := OverallStationStatus.eHoming;
	eCycleControlState.eReady,eCycleControlState.eAutoRun,eCycleControlState.eStartStop:
	    IF (CycleStopReq) THEN
			Status.StationStauts[MM_CONST.CYCLE_CONTROL_HMI_STATE] := OverallStationStatus.eCycleStop;
        ELSE 
			Status.StationStauts[MM_CONST.CYCLE_CONTROL_HMI_STATE] := OverallStationStatus.eRunning;	
		END_IF
	    
	eCycleControlState.eWaitForHomingAfterEStop:
	    IF (GVL_IO.MC_XAirPressureOK AND GVL_IO.MC_NotEStopped) THEN
	         Status.StationStauts[MM_CONST.CYCLE_CONTROL_HMI_STATE] := OverallStationStatus.eHoming;
	    ELSE 
			Status.StationStauts[MM_CONST.CYCLE_CONTROL_HMI_STATE] := OverallStationStatus.eCycleStop;
		END_IF   
		
	ELSE;	
END_CASE
END_METHOD

METHOD PUBLIC ResetCycleControlState : BOOL
VAR_INPUT
END_VAR
State:= eCycleControlState.eUnknown;
NextState:= eCycleControlState.eUnknown;
CycleStopReq := FALSE;
END_METHOD

ACTION StackLightGreen:
GVL_IO.MC_YStackLightRed := FALSE;
GVL_IO.MC_YStackLightYellow := FALSE;
GVL_IO.MC_YStackLightGreen := TRUE;
END_ACTION

ACTION StackLightRed:
GVL_IO.MC_YStackLightRed := TRUE;
GVL_IO.MC_YStackLightYellow := FALSE;
GVL_IO.MC_YStackLightGreen := FALSE;
END_ACTION

ACTION StackLightYellow:
GVL_IO.MC_YStackLightRed := FALSE;
GVL_IO.MC_YStackLightYellow := TRUE;
GVL_IO.MC_YStackLightGreen := FALSE;
END_ACTION

